METHOD PUBLIC Check_DT_TO_DINT_Max
VAR
	value : DT := DatatypeLimits.MAX_VALUE_OF_DT_WHICH_CAN_BE_HELD_IN_A_DINT;
	actual : DINT;
	converted : BOOL;
	equal : BOOL;
END_VAR
TEST('Check_DT_TO_DINT_Max');

// @TEST-RUN
converted := TryConvert_DT_TO_Destination(value, actual);
equal := actual = DT_TO_DINT(value);

// @TEST-ASSERT
AssertTrue(Condition := equal, Message := 'Did not convert DT to DINT correctly');
AssertTrue(Condition := converted, Message := 'Did not report DT to DINT conversion was successful');

TEST_FINISHED();
END_METHOD

METHOD PUBLIC Check_DT_TO_DINT_Min
VAR
	value : DT := DatatypeLimits.DT_MIN_VALUE;
	actual : DINT;
	converted : BOOL;
	equal : BOOL;
END_VAR
TEST('Check_DT_TO_DINT_Min');

// @TEST-RUN
converted := TryConvert_DT_TO_Destination(value, actual);
equal := actual = DT_TO_DINT(value);

// @TEST-ASSERT
AssertTrue(Condition := equal, Message := 'Did not convert DT to DINT correctly');
AssertTrue(Condition := converted, Message := 'Did not report DT to DINT conversion was successful');

TEST_FINISHED();
END_METHOD

METHOD PUBLIC Check_DT_TO_DINT_TooHigh
VAR
	value : DT := DatatypeLimits.DT_MAX_VALUE;
	actual : DINT;
	converted : BOOL;
END_VAR
TEST('Check_DT_TO_DINT_TooHigh');

// @TEST-RUN
converted := TryConvert_DT_TO_Destination(value, actual);

// @TEST-ASSERT
AssertFalse(Condition := converted, Message := 'Did not report DT to DINT conversion was prevented');

TEST_FINISHED();
END_METHOD

METHOD PUBLIC Check_DT_TO_DT_Max
VAR
	value : DT := DatatypeLimits.DT_MAX_VALUE;
	actual : DT;
	converted : BOOL;
	equal : BOOL;
END_VAR
TEST('Check_DT_TO_DT_Max');

// @TEST-RUN
converted := TryConvert_DT_TO_Destination(value, actual);
equal := actual = value;

// @TEST-ASSERT
AssertTrue(Condition := equal, Message := 'Did not convert DT to DT correctly');
AssertTrue(Condition := converted, Message := 'Did not report DT to DT conversion was successful');

TEST_FINISHED();
END_METHOD

METHOD PUBLIC Check_DT_TO_DT_Min
VAR
	value : DT := DatatypeLimits.DT_MIN_VALUE;
	actual : DT;
	converted : BOOL;
	equal : BOOL;
END_VAR
TEST('Check_DT_TO_DT_Min');

// @TEST-RUN
converted := TryConvert_DT_TO_Destination(value, actual);
equal := actual = value;

// @TEST-ASSERT
AssertTrue(Condition := equal, Message := 'Did not convert DT to DT correctly');
AssertTrue(Condition := converted, Message := 'Did not report DT to DT conversion was successful');

TEST_FINISHED();
END_METHOD

METHOD PUBLIC Check_DT_TO_DWORD_Max
VAR
	value : DT := DatatypeLimits.DT_MAX_VALUE;
	actual : DWORD;
	converted : BOOL;
	equal : BOOL;
END_VAR
TEST('Check_DT_TO_DWORD_Max');

// @TEST-RUN
converted := TryConvert_DT_TO_Destination(value, actual);
equal := actual = DT_TO_DWORD(value);

// @TEST-ASSERT
AssertTrue(Condition := equal, Message := 'Did not convert DT to DWORD correctly');
AssertTrue(Condition := converted, Message := 'Did not report DT to DWORD conversion was successful');

TEST_FINISHED();
END_METHOD

METHOD PUBLIC Check_DT_TO_DWORD_Min
VAR
	value : DT := DatatypeLimits.DT_MIN_VALUE;
	actual : DWORD;
	converted : BOOL;
	equal : BOOL;
END_VAR
TEST('Check_DT_TO_DWORD_Min');

// @TEST-RUN
converted := TryConvert_DT_TO_Destination(value, actual);
equal := actual = DT_TO_DWORD(value);

// @TEST-ASSERT
AssertTrue(Condition := equal, Message := 'Did not convert DT to DWORD correctly');
AssertTrue(Condition := converted, Message := 'Did not report DT to DWORD conversion was successful');

TEST_FINISHED();
END_METHOD

METHOD PUBLIC Check_DT_TO_INT_Max
VAR
	value : DT := DatatypeLimits.MAX_VALUE_OF_DT_WHICH_CAN_BE_HELD_IN_A_INT;
	actual : INT;
	converted : BOOL;
	equal : BOOL;
END_VAR
TEST('Check_DT_TO_INT_Max');

// @TEST-RUN
converted := TryConvert_DT_TO_Destination(value, actual);
equal := actual = DT_TO_INT(value);

// @TEST-ASSERT
AssertTrue(Condition := equal, Message := 'Did not convert DT to INT correctly');
AssertTrue(Condition := converted, Message := 'Did not report DT to INT conversion was successful');

TEST_FINISHED();
END_METHOD

METHOD PUBLIC Check_DT_TO_INT_Min
VAR
	value : DT := DatatypeLimits.DT_MIN_VALUE;
	actual : INT;
	converted : BOOL;
	equal : BOOL;
END_VAR
TEST('Check_DT_TO_INT_Min');

// @TEST-RUN
converted := TryConvert_DT_TO_Destination(value, actual);
equal := actual = DT_TO_INT(value);

// @TEST-ASSERT
AssertTrue(Condition := equal, Message := 'Did not convert DT to INT correctly');
AssertTrue(Condition := converted, Message := 'Did not report DT to INT conversion was successful');

TEST_FINISHED();
END_METHOD

METHOD PUBLIC Check_DT_TO_INT_TooHigh
VAR
	value : DT := DatatypeLimits.DT_MAX_VALUE;
	actual : INT;
	converted : BOOL;
END_VAR
TEST('Check_DT_TO_INT_TooHigh');

// @TEST-RUN
converted := TryConvert_DT_TO_Destination(value, actual);

// @TEST-ASSERT
AssertFalse(Condition := converted, Message := 'Did not report DT to INT conversion was prevented');

TEST_FINISHED();
END_METHOD

METHOD PUBLIC Check_DT_TO_LINT_Max
VAR
	value : DT := DatatypeLimits.DT_MAX_VALUE;
	actual : LINT;
	converted : BOOL;
	equal : BOOL;
END_VAR
TEST('Check_DT_TO_LINT_Max');

// @TEST-RUN
converted := TryConvert_DT_TO_Destination(value, actual);
equal := actual = DT_TO_LINT(value);

// @TEST-ASSERT
AssertTrue(Condition := equal, Message := 'Did not convert DT to LINT correctly');
AssertTrue(Condition := converted, Message := 'Did not report DT to LINT conversion was successful');

TEST_FINISHED();
END_METHOD

METHOD PUBLIC Check_DT_TO_LINT_Min
VAR
	value : DT := DatatypeLimits.DT_MIN_VALUE;
	actual : LINT;
	converted : BOOL;
	equal : BOOL;
END_VAR
TEST('Check_DT_TO_LINT_Min');

// @TEST-RUN
converted := TryConvert_DT_TO_Destination(value, actual);
equal := actual = DT_TO_LINT(value);

// @TEST-ASSERT
AssertTrue(Condition := equal, Message := 'Did not convert DT to LINT correctly');
AssertTrue(Condition := converted, Message := 'Did not report DT to LINT conversion was successful');

TEST_FINISHED();
END_METHOD

METHOD PUBLIC Check_DT_TO_LREAL_Max
VAR
	value : DT := DatatypeLimits.DT_MAX_VALUE;
	actual : LREAL;
	converted : BOOL;
	equal : BOOL;
END_VAR
TEST('Check_DT_TO_LREAL_Max');

// @TEST-RUN
converted := TryConvert_DT_TO_Destination(value, actual);
equal := actual = DT_TO_LREAL(value);

// @TEST-ASSERT
AssertTrue(Condition := equal, Message := 'Did not convert DT to LREAL correctly');
AssertTrue(Condition := converted, Message := 'Did not report DT to LREAL conversion was successful');

TEST_FINISHED();
END_METHOD

METHOD PUBLIC Check_DT_TO_LREAL_Min
VAR
	value : DT := DatatypeLimits.DT_MIN_VALUE;
	actual : LREAL;
	converted : BOOL;
	equal : BOOL;
END_VAR
TEST('Check_DT_TO_LREAL_Min');

// @TEST-RUN
converted := TryConvert_DT_TO_Destination(value, actual);
equal := actual = DT_TO_LREAL(value);

// @TEST-ASSERT
AssertTrue(Condition := equal, Message := 'Did not convert DT to LREAL correctly');
AssertTrue(Condition := converted, Message := 'Did not report DT to LREAL conversion was successful');

TEST_FINISHED();
END_METHOD

METHOD PUBLIC Check_DT_TO_LWORD_Max
VAR
	value : DT := DatatypeLimits.DT_MAX_VALUE;
	actual : LWORD;
	converted : BOOL;
	equal : BOOL;
END_VAR
TEST('Check_DT_TO_LWORD_Max');

// @TEST-RUN
converted := TryConvert_DT_TO_Destination(value, actual);
equal := actual = DT_TO_LWORD(value);

// @TEST-ASSERT
AssertTrue(Condition := equal, Message := 'Did not convert DT to LWORD correctly');
AssertTrue(Condition := converted, Message := 'Did not report DT to LWORD conversion was successful');

TEST_FINISHED();
END_METHOD

METHOD PUBLIC Check_DT_TO_LWORD_Min
VAR
	value : DT := DatatypeLimits.DT_MIN_VALUE;
	actual : LWORD;
	converted : BOOL;
	equal : BOOL;
END_VAR
TEST('Check_DT_TO_LWORD_Min');

// @TEST-RUN
converted := TryConvert_DT_TO_Destination(value, actual);
equal := actual = DT_TO_LWORD(value);

// @TEST-ASSERT
AssertTrue(Condition := equal, Message := 'Did not convert DT to LWORD correctly');
AssertTrue(Condition := converted, Message := 'Did not report DT to LWORD conversion was successful');

TEST_FINISHED();
END_METHOD

METHOD PUBLIC Check_DT_TO_REAL_Max
VAR
	value : DT := DatatypeLimits.DT_MAX_VALUE;
	actual : REAL;
	converted : BOOL;
	equal : BOOL;
END_VAR
TEST('Check_DT_TO_REAL_Max');

// @TEST-RUN
converted := TryConvert_DT_TO_Destination(value, actual);
equal := actual = DT_TO_REAL(value);

// @TEST-ASSERT
AssertTrue(Condition := equal, Message := 'Did not convert DT to REAL correctly');
AssertTrue(Condition := converted, Message := 'Did not report DT to REAL conversion was successful');

TEST_FINISHED();
END_METHOD

METHOD PUBLIC Check_DT_TO_REAL_Min
VAR
	value : DT := DatatypeLimits.DT_MIN_VALUE;
	actual : REAL;
	converted : BOOL;
	equal : BOOL;
END_VAR
TEST('Check_DT_TO_REAL_Min');

// @TEST-RUN
converted := TryConvert_DT_TO_Destination(value, actual);
equal := actual = DT_TO_REAL(value);

// @TEST-ASSERT
AssertTrue(Condition := equal, Message := 'Did not convert DT to REAL correctly');
AssertTrue(Condition := converted, Message := 'Did not report DT to REAL conversion was successful');

TEST_FINISHED();
END_METHOD

METHOD PUBLIC Check_DT_TO_SINT_Max
VAR
	value : DT := DatatypeLimits.MAX_VALUE_OF_DT_WHICH_CAN_BE_HELD_IN_A_SINT;
	actual : SINT;
	converted : BOOL;
	equal : BOOL;
END_VAR
TEST('Check_DT_TO_SINT_Max');

// @TEST-RUN
converted := TryConvert_DT_TO_Destination(value, actual);
equal := actual = DT_TO_SINT(value);

// @TEST-ASSERT
AssertTrue(Condition := equal, Message := 'Did not convert DT to SINT correctly');
AssertTrue(Condition := converted, Message := 'Did not report DT to SINT conversion was successful');

TEST_FINISHED();
END_METHOD

METHOD PUBLIC Check_DT_TO_SINT_Min
VAR
	value : DT := DatatypeLimits.DT_MIN_VALUE;
	actual : SINT;
	converted : BOOL;
	equal : BOOL;
END_VAR
TEST('Check_DT_TO_SINT_Min');

// @TEST-RUN
converted := TryConvert_DT_TO_Destination(value, actual);
equal := actual = DT_TO_SINT(value);

// @TEST-ASSERT
AssertTrue(Condition := equal, Message := 'Did not convert DT to SINT correctly');
AssertTrue(Condition := converted, Message := 'Did not report DT to SINT conversion was successful');

TEST_FINISHED();
END_METHOD

METHOD PUBLIC Check_DT_TO_SINT_TooHigh
VAR
	value : DT := DatatypeLimits.DT_MAX_VALUE;
	actual : SINT;
	converted : BOOL;
END_VAR
TEST('Check_DT_TO_SINT_TooHigh');

// @TEST-RUN
converted := TryConvert_DT_TO_Destination(value, actual);

// @TEST-ASSERT
AssertFalse(Condition := converted, Message := 'Did not report DT to SINT conversion was prevented');

TEST_FINISHED();
END_METHOD

METHOD PUBLIC Check_DT_TO_STRING_Max
VAR
	value : DT := DatatypeLimits.DT_MAX_VALUE;
	actual : STRING;
	converted : BOOL;
	equal : BOOL;
END_VAR
TEST('Check_DT_TO_STRING_Max');

// @TEST-RUN
converted := TryConvert_DT_TO_Destination(value, actual);
equal := actual = DT_TO_STRING(value);

// @TEST-ASSERT
AssertTrue(Condition := equal, Message := 'Did not convert DT to STRING correctly');
AssertTrue(Condition := converted, Message := 'Did not report DT to STRING conversion was successful');

TEST_FINISHED();
END_METHOD

METHOD PUBLIC Check_DT_TO_STRING_Min
VAR
	value : DT := DatatypeLimits.DT_MIN_VALUE;
	actual : STRING;
	converted : BOOL;
	equal : BOOL;
END_VAR
TEST('Check_DT_TO_STRING_Min');

// @TEST-RUN
converted := TryConvert_DT_TO_Destination(value, actual);
equal := actual = DT_TO_STRING(value);

// @TEST-ASSERT
AssertTrue(Condition := equal, Message := 'Did not convert DT to STRING correctly');
AssertTrue(Condition := converted, Message := 'Did not report DT to STRING conversion was successful');

TEST_FINISHED();
END_METHOD

METHOD PUBLIC Check_DT_TO_TIME_Max
VAR
	value : DT := DatatypeLimits.MAX_VALUE_OF_DT_WHICH_CAN_BE_HELD_IN_A_TIME;
	actual : TIME;
	converted : BOOL;
	equal : BOOL;
END_VAR
TEST('Check_DT_TO_TIME_Max');

// @TEST-RUN
converted := TryConvert_DT_TO_Destination(value, actual);
equal := actual = DT_TO_TIME(value);

// @TEST-ASSERT
AssertTrue(Condition := equal, Message := 'Did not convert DT to TIME correctly');
AssertTrue(Condition := converted, Message := 'Did not report DT to TIME conversion was successful');

TEST_FINISHED();
END_METHOD

METHOD PUBLIC Check_DT_TO_TIME_Min
VAR
	value : DT := DatatypeLimits.DT_MIN_VALUE;
	actual : TIME;
	converted : BOOL;
	equal : BOOL;
END_VAR
TEST('Check_DT_TO_TIME_Min');

// @TEST-RUN
converted := TryConvert_DT_TO_Destination(value, actual);
equal := actual = DT_TO_TIME(value);

// @TEST-ASSERT
AssertTrue(Condition := equal, Message := 'Did not convert DT to TIME correctly');
AssertTrue(Condition := converted, Message := 'Did not report DT to TIME conversion was successful');

TEST_FINISHED();
END_METHOD

METHOD PUBLIC Check_DT_TO_TIME_TooHigh
VAR
	value : DT := DatatypeLimits.DT_MAX_VALUE;
	actual : TIME;
	converted : BOOL;
END_VAR
TEST('Check_DT_TO_TIME_TooHigh');

// @TEST-RUN
converted := TryConvert_DT_TO_Destination(value, actual);

// @TEST-ASSERT
AssertFalse(Condition := converted, Message := 'Did not report DT to TIME conversion was prevented');

TEST_FINISHED();
END_METHOD

METHOD PUBLIC Check_DT_TO_TOD_Max
VAR
	value : DT := DatatypeLimits.MAX_VALUE_OF_DT_WHICH_CAN_BE_HELD_IN_A_TOD;
	actual : TOD;
	converted : BOOL;
	equal : BOOL;
END_VAR
TEST('Check_DT_TO_TOD_Max');

// @TEST-RUN
converted := TryConvert_DT_TO_Destination(value, actual);
equal := actual = DT_TO_TOD(value);

// @TEST-ASSERT
AssertTrue(Condition := equal, Message := 'Did not convert DT to TOD correctly');
AssertTrue(Condition := converted, Message := 'Did not report DT to TOD conversion was successful');

TEST_FINISHED();
END_METHOD

METHOD PUBLIC Check_DT_TO_TOD_Min
VAR
	value : DT := DatatypeLimits.DT_MIN_VALUE;
	actual : TOD;
	converted : BOOL;
	equal : BOOL;
END_VAR
TEST('Check_DT_TO_TOD_Min');

// @TEST-RUN
converted := TryConvert_DT_TO_Destination(value, actual);
equal := actual = DT_TO_TOD(value);

// @TEST-ASSERT
AssertTrue(Condition := equal, Message := 'Did not convert DT to TOD correctly');
AssertTrue(Condition := converted, Message := 'Did not report DT to TOD conversion was successful');

TEST_FINISHED();
END_METHOD

METHOD PUBLIC Check_DT_TO_TOD_TooHigh
VAR
	value : DT := DatatypeLimits.DT_MAX_VALUE;
	actual : TOD;
	converted : BOOL;
END_VAR
TEST('Check_DT_TO_TOD_TooHigh');

// @TEST-RUN
converted := TryConvert_DT_TO_Destination(value, actual);

// @TEST-ASSERT
AssertFalse(Condition := converted, Message := 'Did not report DT to TOD conversion was prevented');

TEST_FINISHED();
END_METHOD

METHOD PUBLIC Check_DT_TO_UDINT_Max
VAR
	value : DT := DatatypeLimits.DT_MAX_VALUE;
	actual : UDINT;
	converted : BOOL;
	equal : BOOL;
END_VAR
TEST('Check_DT_TO_UDINT_Max');

// @TEST-RUN
converted := TryConvert_DT_TO_Destination(value, actual);
equal := actual = DT_TO_UDINT(value);

// @TEST-ASSERT
AssertTrue(Condition := equal, Message := 'Did not convert DT to UDINT correctly');
AssertTrue(Condition := converted, Message := 'Did not report DT to UDINT conversion was successful');

TEST_FINISHED();
END_METHOD

METHOD PUBLIC Check_DT_TO_UDINT_Min
VAR
	value : DT := DatatypeLimits.DT_MIN_VALUE;
	actual : UDINT;
	converted : BOOL;
	equal : BOOL;
END_VAR
TEST('Check_DT_TO_UDINT_Min');

// @TEST-RUN
converted := TryConvert_DT_TO_Destination(value, actual);
equal := actual = DT_TO_UDINT(value);

// @TEST-ASSERT
AssertTrue(Condition := equal, Message := 'Did not convert DT to UDINT correctly');
AssertTrue(Condition := converted, Message := 'Did not report DT to UDINT conversion was successful');

TEST_FINISHED();
END_METHOD

METHOD PUBLIC Check_DT_TO_UINT_Max
VAR
	value : DT := DatatypeLimits.MAX_VALUE_OF_DT_WHICH_CAN_BE_HELD_IN_A_UINT;
	actual : UINT;
	converted : BOOL;
	equal : BOOL;
END_VAR
TEST('Check_DT_TO_UINT_Max');

// @TEST-RUN
converted := TryConvert_DT_TO_Destination(value, actual);
equal := actual = DT_TO_UINT(value);

// @TEST-ASSERT
AssertTrue(Condition := equal, Message := 'Did not convert DT to UINT correctly');
AssertTrue(Condition := converted, Message := 'Did not report DT to UINT conversion was successful');

TEST_FINISHED();
END_METHOD

METHOD PUBLIC Check_DT_TO_UINT_Min
VAR
	value : DT := DatatypeLimits.DT_MIN_VALUE;
	actual : UINT;
	converted : BOOL;
	equal : BOOL;
END_VAR
TEST('Check_DT_TO_UINT_Min');

// @TEST-RUN
converted := TryConvert_DT_TO_Destination(value, actual);
equal := actual = DT_TO_UINT(value);

// @TEST-ASSERT
AssertTrue(Condition := equal, Message := 'Did not convert DT to UINT correctly');
AssertTrue(Condition := converted, Message := 'Did not report DT to UINT conversion was successful');

TEST_FINISHED();
END_METHOD

METHOD PUBLIC Check_DT_TO_UINT_TooHigh
VAR
	value : DT := DatatypeLimits.DT_MAX_VALUE;
	actual : UINT;
	converted : BOOL;
END_VAR
TEST('Check_DT_TO_UINT_TooHigh');

// @TEST-RUN
converted := TryConvert_DT_TO_Destination(value, actual);

// @TEST-ASSERT
AssertFalse(Condition := converted, Message := 'Did not report DT to UINT conversion was prevented');

TEST_FINISHED();
END_METHOD

METHOD PUBLIC Check_DT_TO_ULINT_Max
VAR
	value : DT := DatatypeLimits.DT_MAX_VALUE;
	actual : ULINT;
	converted : BOOL;
	equal : BOOL;
END_VAR
TEST('Check_DT_TO_ULINT_Max');

// @TEST-RUN
converted := TryConvert_DT_TO_Destination(value, actual);
equal := actual = DT_TO_ULINT(value);

// @TEST-ASSERT
AssertTrue(Condition := equal, Message := 'Did not convert DT to ULINT correctly');
AssertTrue(Condition := converted, Message := 'Did not report DT to ULINT conversion was successful');

TEST_FINISHED();
END_METHOD

METHOD PUBLIC Check_DT_TO_ULINT_Min
VAR
	value : DT := DatatypeLimits.DT_MIN_VALUE;
	actual : ULINT;
	converted : BOOL;
	equal : BOOL;
END_VAR
TEST('Check_DT_TO_ULINT_Min');

// @TEST-RUN
converted := TryConvert_DT_TO_Destination(value, actual);
equal := actual = DT_TO_ULINT(value);

// @TEST-ASSERT
AssertTrue(Condition := equal, Message := 'Did not convert DT to ULINT correctly');
AssertTrue(Condition := converted, Message := 'Did not report DT to ULINT conversion was successful');

TEST_FINISHED();
END_METHOD

METHOD PUBLIC Check_DT_TO_USINT_Max
VAR
	value : DT := DatatypeLimits.MAX_VALUE_OF_DT_WHICH_CAN_BE_HELD_IN_A_USINT;
	actual : USINT;
	converted : BOOL;
	equal : BOOL;
END_VAR
TEST('Check_DT_TO_USINT_Max');

// @TEST-RUN
converted := TryConvert_DT_TO_Destination(value, actual);
equal := actual = DT_TO_USINT(value);

// @TEST-ASSERT
AssertTrue(Condition := equal, Message := 'Did not convert DT to USINT correctly');
AssertTrue(Condition := converted, Message := 'Did not report DT to USINT conversion was successful');

TEST_FINISHED();
END_METHOD

METHOD PUBLIC Check_DT_TO_USINT_Min
VAR
	value : DT := DatatypeLimits.DT_MIN_VALUE;
	actual : USINT;
	converted : BOOL;
	equal : BOOL;
END_VAR
TEST('Check_DT_TO_USINT_Min');

// @TEST-RUN
converted := TryConvert_DT_TO_Destination(value, actual);
equal := actual = DT_TO_USINT(value);

// @TEST-ASSERT
AssertTrue(Condition := equal, Message := 'Did not convert DT to USINT correctly');
AssertTrue(Condition := converted, Message := 'Did not report DT to USINT conversion was successful');

TEST_FINISHED();
END_METHOD

METHOD PUBLIC Check_DT_TO_USINT_TooHigh
VAR
	value : DT := DatatypeLimits.DT_MAX_VALUE;
	actual : USINT;
	converted : BOOL;
END_VAR
TEST('Check_DT_TO_USINT_TooHigh');

// @TEST-RUN
converted := TryConvert_DT_TO_Destination(value, actual);

// @TEST-ASSERT
AssertFalse(Condition := converted, Message := 'Did not report DT to USINT conversion was prevented');

TEST_FINISHED();
END_METHOD

METHOD PUBLIC Check_DT_TO_WORD_Max
VAR
	value : DT := DatatypeLimits.MAX_VALUE_OF_DT_WHICH_CAN_BE_HELD_IN_A_WORD;
	actual : WORD;
	converted : BOOL;
	equal : BOOL;
END_VAR
TEST('Check_DT_TO_WORD_Max');

// @TEST-RUN
converted := TryConvert_DT_TO_Destination(value, actual);
equal := actual = DT_TO_WORD(value);

// @TEST-ASSERT
AssertTrue(Condition := equal, Message := 'Did not convert DT to WORD correctly');
AssertTrue(Condition := converted, Message := 'Did not report DT to WORD conversion was successful');

TEST_FINISHED();
END_METHOD

METHOD PUBLIC Check_DT_TO_WORD_Min
VAR
	value : DT := DatatypeLimits.DT_MIN_VALUE;
	actual : WORD;
	converted : BOOL;
	equal : BOOL;
END_VAR
TEST('Check_DT_TO_WORD_Min');

// @TEST-RUN
converted := TryConvert_DT_TO_Destination(value, actual);
equal := actual = DT_TO_WORD(value);

// @TEST-ASSERT
AssertTrue(Condition := equal, Message := 'Did not convert DT to WORD correctly');
AssertTrue(Condition := converted, Message := 'Did not report DT to WORD conversion was successful');

TEST_FINISHED();
END_METHOD

METHOD PUBLIC Check_DT_TO_WORD_TooHigh
VAR
	value : DT := DatatypeLimits.DT_MAX_VALUE;
	actual : WORD;
	converted : BOOL;
END_VAR
TEST('Check_DT_TO_WORD_TooHigh');

// @TEST-RUN
converted := TryConvert_DT_TO_Destination(value, actual);

// @TEST-ASSERT
AssertFalse(Condition := converted, Message := 'Did not report DT to WORD conversion was prevented');

TEST_FINISHED();
END_METHOD

END_FUNCTION_BLOCK

// ---- mobject-converters/Tests/DWORD_TO_TestSuite.TcPOU
FUNCTION_BLOCK PUBLIC DWORD_TO_TestSuite EXTENDS TcUnit.FB_TestSuite
VAR
END_VAR

Check_DWORD_TO_BOOL_Max();
Check_DWORD_TO_BOOL_Min();
Check_DWORD_TO_BYTE_Max();
Check_DWORD_TO_BYTE_Min();
Check_DWORD_TO_BYTE_TooHigh();
Check_DWORD_TO_WORD_Max();
Check_DWORD_TO_WORD_Min();
Check_DWORD_TO_WORD_TooHigh();
Check_DWORD_TO_DWORD_Max();
Check_DWORD_TO_DWORD_Min();
Check_DWORD_TO_LWORD_Max();
Check_DWORD_TO_LWORD_Min();
Check_DWORD_TO_SINT_Max();
Check_DWORD_TO_SINT_Min();
Check_DWORD_TO_SINT_TooHigh();
Check_DWORD_TO_INT_Max();
Check_DWORD_TO_INT_Min();
Check_DWORD_TO_INT_TooHigh();
Check_DWORD_TO_DINT_Max();
Check_DWORD_TO_DINT_Min();
Check_DWORD_TO_DINT_TooHigh();
Check_DWORD_TO_LINT_Max();
Check_DWORD_TO_LINT_Min();
Check_DWORD_TO_USINT_Max();
Check_DWORD_TO_USINT_Min();
Check_DWORD_TO_USINT_TooHigh();
Check_DWORD_TO_UINT_Max();
Check_DWORD_TO_UINT_Min();
Check_DWORD_TO_UINT_TooHigh();
Check_DWORD_TO_UDINT_Max();
Check_DWORD_TO_UDINT_Min();
Check_DWORD_TO_ULINT_Max();
Check_DWORD_TO_ULINT_Min();
Check_DWORD_TO_REAL_Max();
Check_DWORD_TO_REAL_Min();
Check_DWORD_TO_LREAL_Max();
Check_DWORD_TO_LREAL_Min();
Check_DWORD_TO_TIME_Max();
Check_DWORD_TO_TIME_Min();
Check_DWORD_TO_TOD_Max();
Check_DWORD_TO_TOD_Min();
Check_DWORD_TO_TOD_TooHigh();
Check_DWORD_TO_DATE_Max();
Check_DWORD_TO_DATE_Min();
Check_DWORD_TO_DT_Max();
Check_DWORD_TO_DT_Min();
Check_DWORD_TO_STRING_Max();
Check_DWORD_TO_STRING_Min();

METHOD PUBLIC Check_DWORD_TO_BOOL_Max
VAR
	value : DWORD := DatatypeLimits.DWORD_MAX_VALUE;
	actual : BOOL;
	converted : BOOL;
	equal : BOOL;
END_VAR
TEST('Check_DWORD_TO_BOOL_Max');

// @TEST-RUN
converted := TryConvert_DWORD_TO_Destination(value, actual);
equal := actual = DWORD_TO_BOOL(value);

// @TEST-ASSERT
AssertTrue(Condition := equal, Message := 'Did not convert DWORD to BOOL correctly');
AssertTrue(Condition := converted, Message := 'Did not report DWORD to BOOL conversion was successful');

TEST_FINISHED();
END_METHOD

METHOD PUBLIC Check_DWORD_TO_BOOL_Min
VAR
	value : DWORD := DatatypeLimits.DWORD_MIN_VALUE;
	actual : BOOL;
	converted : BOOL;
	equal : BOOL;
END_VAR
TEST('Check_DWORD_TO_BOOL_Min');

// @TEST-RUN
converted := TryConvert_DWORD_TO_Destination(value, actual);
equal := actual = DWORD_TO_BOOL(value);

// @TEST-ASSERT
AssertTrue(Condition := equal, Message := 'Did not convert DWORD to BOOL correctly');
AssertTrue(Condition := converted, Message := 'Did not report DWORD to BOOL conversion was successful');

TEST_FINISHED();
END_METHOD

METHOD PUBLIC Check_DWORD_TO_BYTE_Max
VAR
	value : DWORD := DatatypeLimits.MAX_VALUE_OF_DWORD_WHICH_CAN_BE_HELD_IN_A_BYTE;
	actual : BYTE;
	converted : BOOL;
	equal : BOOL;
END_VAR
TEST('Check_DWORD_TO_BYTE_Max');

// @TEST-RUN
converted := TryConvert_DWORD_TO_Destination(value, actual);
equal := actual = DWORD_TO_BYTE(value);

// @TEST-ASSERT
AssertTrue(Condition := equal, Message := 'Did not convert DWORD to BYTE correctly');
AssertTrue(Condition := converted, Message := 'Did not report DWORD to BYTE conversion was successful');

TEST_FINISHED();
END_METHOD

METHOD PUBLIC Check_DWORD_TO_BYTE_Min
VAR
	value : DWORD := DatatypeLimits.DWORD_MIN_VALUE;
	actual : BYTE;
	converted : BOOL;
	equal : BOOL;
END_VAR
TEST('Check_DWORD_TO_BYTE_Min');

// @TEST-RUN
converted := TryConvert_DWORD_TO_Destination(value, actual);
equal := actual = DWORD_TO_BYTE(value);

// @TEST-ASSERT
AssertTrue(Condition := equal, Message := 'Did not convert DWORD to BYTE correctly');
AssertTrue(Condition := converted, Message := 'Did not report DWORD to BYTE conversion was successful');

TEST_FINISHED();
END_METHOD

METHOD PUBLIC Check_DWORD_TO_BYTE_TooHigh
VAR
	value : DWORD := DatatypeLimits.DWORD_MAX_VALUE;
	actual : BYTE;
	converted : BOOL;
END_VAR
TEST('Check_DWORD_TO_BYTE_TooHigh');

// @TEST-RUN
converted := TryConvert_DWORD_TO_Destination(value, actual);

// @TEST-ASSERT
AssertFalse(Condition := converted, Message := 'Did not report DWORD to BYTE conversion was prevented');

TEST_FINISHED();
END_METHOD

METHOD PUBLIC Check_DWORD_TO_DATE_Max
VAR
	value : DWORD := DatatypeLimits.DWORD_MAX_VALUE;
	actual : DATE;
	converted : BOOL;
	equal : BOOL;
END_VAR
TEST('Check_DWORD_TO_DATE_Max');

// @TEST-RUN
converted := TryConvert_DWORD_TO_Destination(value, actual);
equal := actual = DWORD_TO_DATE(value);

// @TEST-ASSERT
AssertTrue(Condition := equal, Message := 'Did not convert DWORD to DATE correctly');
AssertTrue(Condition := converted, Message := 'Did not report DWORD to DATE conversion was successful');

TEST_FINISHED();
END_METHOD

METHOD PUBLIC Check_DWORD_TO_DATE_Min
VAR
	value : DWORD := DatatypeLimits.DWORD_MIN_VALUE;
	actual : DATE;
	converted : BOOL;
	equal : BOOL;
END_VAR
TEST('Check_DWORD_TO_DATE_Min');

// @TEST-RUN
converted := TryConvert_DWORD_TO_Destination(value, actual);
equal := actual = DWORD_TO_DATE(value);

// @TEST-ASSERT
AssertTrue(Condition := equal, Message := 'Did not convert DWORD to DATE correctly');
AssertTrue(Condition := converted, Message := 'Did not report DWORD to DATE conversion was successful');

TEST_FINISHED();
END_METHOD

METHOD PUBLIC Check_DWORD_TO_DINT_Max
VAR
	value : DWORD := DatatypeLimits.MAX_VALUE_OF_DWORD_WHICH_CAN_BE_HELD_IN_A_DINT;
	actual : DINT;
	converted : BOOL;
	equal : BOOL;
END_VAR
TEST('Check_DWORD_TO_DINT_Max');

// @TEST-RUN
converted := TryConvert_DWORD_TO_Destination(value, actual);
equal := actual = DWORD_TO_DINT(value);

// @TEST-ASSERT
AssertTrue(Condition := equal, Message := 'Did not convert DWORD to DINT correctly');
AssertTrue(Condition := converted, Message := 'Did not report DWORD to DINT conversion was successful');

TEST_FINISHED();
END_METHOD

METHOD PUBLIC Check_DWORD_TO_DINT_Min
VAR
	value : DWORD := DatatypeLimits.DWORD_MIN_VALUE;
	actual : DINT;
	converted : BOOL;
	equal : BOOL;
END_VAR
TEST('Check_DWORD_TO_DINT_Min');

// @TEST-RUN
converted := TryConvert_DWORD_TO_Destination(value, actual);
equal := actual = DWORD_TO_DINT(value);

// @TEST-ASSERT
AssertTrue(Condition := equal, Message := 'Did not convert DWORD to DINT correctly');
AssertTrue(Condition := converted, Message := 'Did not report DWORD to DINT conversion was successful');

TEST_FINISHED();
END_METHOD

METHOD PUBLIC Check_DWORD_TO_DINT_TooHigh
VAR
	value : DWORD := DatatypeLimits.DWORD_MAX_VALUE;
	actual : DINT;
	converted : BOOL;
END_VAR
TEST('Check_DWORD_TO_DINT_TooHigh');

// @TEST-RUN
converted := TryConvert_DWORD_TO_Destination(value, actual);

// @TEST-ASSERT
AssertFalse(Condition := converted, Message := 'Did not report DWORD to DINT conversion was prevented');

TEST_FINISHED();
END_METHOD

METHOD PUBLIC Check_DWORD_TO_DT_Max
VAR
	value : DWORD := DatatypeLimits.DWORD_MAX_VALUE;
	actual : DT;
	converted : BOOL;
	equal : BOOL;
END_VAR
TEST('Check_DWORD_TO_DT_Max');

// @TEST-RUN
converted := TryConvert_DWORD_TO_Destination(value, actual);
equal := actual = DWORD_TO_DT(value);

// @TEST-ASSERT
AssertTrue(Condition := equal, Message := 'Did not convert DWORD to DT correctly');
AssertTrue(Condition := converted, Message := 'Did not report DWORD to DT conversion was successful');

TEST_FINISHED();
END_METHOD

METHOD PUBLIC Check_DWORD_TO_DT_Min
VAR
	value : DWORD := DatatypeLimits.DWORD_MIN_VALUE;
	actual : DT;
	converted : BOOL;
	equal : BOOL;
END_VAR
TEST('Check_DWORD_TO_DT_Min');

// @TEST-RUN
converted := TryConvert_DWORD_TO_Destination(value, actual);
equal := actual = DWORD_TO_DT(value);

// @TEST-ASSERT
AssertTrue(Condition := equal, Message := 'Did not convert DWORD to DT correctly');
AssertTrue(Condition := converted, Message := 'Did not report DWORD to DT conversion was successful');

TEST_FINISHED();
END_METHOD

METHOD PUBLIC Check_DWORD_TO_DWORD_Max
VAR
	value : DWORD := DatatypeLimits.DWORD_MAX_VALUE;
	actual : DWORD;
	converted : BOOL;
	equal : BOOL;
END_VAR
TEST('Check_DWORD_TO_DWORD_Max');

// @TEST-RUN
converted := TryConvert_DWORD_TO_Destination(value, actual);
equal := actual = value;

// @TEST-ASSERT
AssertTrue(Condition := equal, Message := 'Did not convert DWORD to DWORD correctly');
AssertTrue(Condition := converted, Message := 'Did not report DWORD to DWORD conversion was successful');

TEST_FINISHED();
END_METHOD

METHOD PUBLIC Check_DWORD_TO_DWORD_Min
VAR
	value : DWORD := DatatypeLimits.DWORD_MIN_VALUE;
	actual : DWORD;
	converted : BOOL;
	equal : BOOL;
END_VAR
TEST('Check_DWORD_TO_DWORD_Min');

// @TEST-RUN
converted := TryConvert_DWORD_TO_Destination(value, actual);
equal := actual = value;

// @TEST-ASSERT
AssertTrue(Condition := equal, Message := 'Did not convert DWORD to DWORD correctly');
AssertTrue(Condition := converted, Message := 'Did not report DWORD to DWORD conversion was successful');

TEST_FINISHED();
END_METHOD

METHOD PUBLIC Check_DWORD_TO_INT_Max
VAR
	value : DWORD := DatatypeLimits.MAX_VALUE_OF_DWORD_WHICH_CAN_BE_HELD_IN_A_INT;
	actual : INT;
	converted : BOOL;
	equal : BOOL;
END_VAR
TEST('Check_DWORD_TO_INT_Max');

// @TEST-RUN
converted := TryConvert_DWORD_TO_Destination(value, actual);
equal := actual = DWORD_TO_INT(value);

// @TEST-ASSERT
AssertTrue(Condition := equal, Message := 'Did not convert DWORD to INT correctly');
AssertTrue(Condition := converted, Message := 'Did not report DWORD to INT conversion was successful');

TEST_FINISHED();
END_METHOD

METHOD PUBLIC Check_DWORD_TO_INT_Min
VAR
	value : DWORD := DatatypeLimits.DWORD_MIN_VALUE;
	actual : INT;
	converted : BOOL;
	equal : BOOL;
END_VAR
TEST('Check_DWORD_TO_INT_Min');

// @TEST-RUN
converted := TryConvert_DWORD_TO_Destination(value, actual);
equal := actual = DWORD_TO_INT(value);

// @TEST-ASSERT
AssertTrue(Condition := equal, Message := 'Did not convert DWORD to INT correctly');
AssertTrue(Condition := converted, Message := 'Did not report DWORD to INT conversion was successful');

TEST_FINISHED();
END_METHOD

METHOD PUBLIC Check_DWORD_TO_INT_TooHigh
VAR
	value : DWORD := DatatypeLimits.DWORD_MAX_VALUE;
	actual : INT;
	converted : BOOL;
END_VAR
TEST('Check_DWORD_TO_INT_TooHigh');

// @TEST-RUN
converted := TryConvert_DWORD_TO_Destination(value, actual);

// @TEST-ASSERT
AssertFalse(Condition := converted, Message := 'Did not report DWORD to INT conversion was prevented');

TEST_FINISHED();
END_METHOD

METHOD PUBLIC Check_DWORD_TO_LINT_Max
VAR
	value : DWORD := DatatypeLimits.DWORD_MAX_VALUE;
	actual : LINT;
	converted : BOOL;
	equal : BOOL;
END_VAR
TEST('Check_DWORD_TO_LINT_Max');

// @TEST-RUN
converted := TryConvert_DWORD_TO_Destination(value, actual);
equal := actual = DWORD_TO_LINT(value);

// @TEST-ASSERT
AssertTrue(Condition := equal, Message := 'Did not convert DWORD to LINT correctly');
AssertTrue(Condition := converted, Message := 'Did not report DWORD to LINT conversion was successful');

TEST_FINISHED();
END_METHOD

METHOD PUBLIC Check_DWORD_TO_LINT_Min
VAR
	value : DWORD := DatatypeLimits.DWORD_MIN_VALUE;
	actual : LINT;
	converted : BOOL;
	equal : BOOL;
END_VAR
TEST('Check_DWORD_TO_LINT_Min');

// @TEST-RUN
converted := TryConvert_DWORD_TO_Destination(value, actual);
equal := actual = DWORD_TO_LINT(value);

// @TEST-ASSERT
AssertTrue(Condition := equal, Message := 'Did not convert DWORD to LINT correctly');
AssertTrue(Condition := converted, Message := 'Did not report DWORD to LINT conversion was successful');

TEST_FINISHED();
END_METHOD

METHOD PUBLIC Check_DWORD_TO_LREAL_Max
VAR
	value : DWORD := DatatypeLimits.DWORD_MAX_VALUE;
	actual : LREAL;
	converted : BOOL;
	equal : BOOL;
END_VAR
TEST('Check_DWORD_TO_LREAL_Max');

// @TEST-RUN
converted := TryConvert_DWORD_TO_Destination(value, actual);
equal := actual = DWORD_TO_LREAL(value);

// @TEST-ASSERT
AssertTrue(Condition := equal, Message := 'Did not convert DWORD to LREAL correctly');
AssertTrue(Condition := converted, Message := 'Did not report DWORD to LREAL conversion was successful');

TEST_FINISHED();
END_METHOD

METHOD PUBLIC Check_DWORD_TO_LREAL_Min
VAR
	value : DWORD := DatatypeLimits.DWORD_MIN_VALUE;
	actual : LREAL;
	converted : BOOL;
	equal : BOOL;
END_VAR
TEST('Check_DWORD_TO_LREAL_Min');

// @TEST-RUN
converted := TryConvert_DWORD_TO_Destination(value, actual);
equal := actual = DWORD_TO_LREAL(value);

// @TEST-ASSERT
AssertTrue(Condition := equal, Message := 'Did not convert DWORD to LREAL correctly');
AssertTrue(Condition := converted, Message := 'Did not report DWORD to LREAL conversion was successful');

TEST_FINISHED();
END_METHOD

METHOD PUBLIC Check_DWORD_TO_LWORD_Max
VAR
	value : DWORD := DatatypeLimits.DWORD_MAX_VALUE;
	actual : LWORD;
	converted : BOOL;
	equal : BOOL;
END_VAR
TEST('Check_DWORD_TO_LWORD_Max');

// @TEST-RUN
converted := TryConvert_DWORD_TO_Destination(value, actual);
equal := actual = DWORD_TO_LWORD(value);

// @TEST-ASSERT
AssertTrue(Condition := equal, Message := 'Did not convert DWORD to LWORD correctly');
AssertTrue(Condition := converted, Message := 'Did not report DWORD to LWORD conversion was successful');

TEST_FINISHED();
END_METHOD

METHOD PUBLIC Check_DWORD_TO_LWORD_Min
VAR
	value : DWORD := DatatypeLimits.DWORD_MIN_VALUE;
	actual : LWORD;
	converted : BOOL;
	equal : BOOL;
END_VAR
TEST('Check_DWORD_TO_LWORD_Min');

// @TEST-RUN
converted := TryConvert_DWORD_TO_Destination(value, actual);
equal := actual = DWORD_TO_LWORD(value);

// @TEST-ASSERT
AssertTrue(Condition := equal, Message := 'Did not convert DWORD to LWORD correctly');
AssertTrue(Condition := converted, Message := 'Did not report DWORD to LWORD conversion was successful');

TEST_FINISHED();
END_METHOD

METHOD PUBLIC Check_DWORD_TO_REAL_Max
VAR
	value : DWORD := DatatypeLimits.DWORD_MAX_VALUE;
	actual : REAL;
	converted : BOOL;
	equal : BOOL;
END_VAR
TEST('Check_DWORD_TO_REAL_Max');

// @TEST-RUN
converted := TryConvert_DWORD_TO_Destination(value, actual);
equal := actual = DWORD_TO_REAL(value);

// @TEST-ASSERT
AssertTrue(Condition := equal, Message := 'Did not convert DWORD to REAL correctly');
AssertTrue(Condition := converted, Message := 'Did not report DWORD to REAL conversion was successful');

TEST_FINISHED();
END_METHOD

METHOD PUBLIC Check_DWORD_TO_REAL_Min
VAR
	value : DWORD := DatatypeLimits.DWORD_MIN_VALUE;
	actual : REAL;
	converted : BOOL;
	equal : BOOL;
END_VAR
TEST('Check_DWORD_TO_REAL_Min');

// @TEST-RUN
converted := TryConvert_DWORD_TO_Destination(value, actual);
equal := actual = DWORD_TO_REAL(value);

// @TEST-ASSERT
AssertTrue(Condition := equal, Message := 'Did not convert DWORD to REAL correctly');
AssertTrue(Condition := converted, Message := 'Did not report DWORD to REAL conversion was successful');

TEST_FINISHED();
END_METHOD

METHOD PUBLIC Check_DWORD_TO_SINT_Max
VAR
	value : DWORD := DatatypeLimits.MAX_VALUE_OF_DWORD_WHICH_CAN_BE_HELD_IN_A_SINT;
	actual : SINT;
	converted : BOOL;
	equal : BOOL;
END_VAR
TEST('Check_DWORD_TO_SINT_Max');

// @TEST-RUN
converted := TryConvert_DWORD_TO_Destination(value, actual);
equal := actual = DWORD_TO_SINT(value);

// @TEST-ASSERT
AssertTrue(Condition := equal, Message := 'Did not convert DWORD to SINT correctly');
AssertTrue(Condition := converted, Message := 'Did not report DWORD to SINT conversion was successful');

TEST_FINISHED();
END_METHOD

METHOD PUBLIC Check_DWORD_TO_SINT_Min
VAR
	value : DWORD := DatatypeLimits.DWORD_MIN_VALUE;
	actual : SINT;
	converted : BOOL;
	equal : BOOL;
END_VAR
TEST('Check_DWORD_TO_SINT_Min');

// @TEST-RUN
converted := TryConvert_DWORD_TO_Destination(value, actual);
equal := actual = DWORD_TO_SINT(value);

// @TEST-ASSERT
AssertTrue(Condition := equal, Message := 'Did not convert DWORD to SINT correctly');
AssertTrue(Condition := converted, Message := 'Did not report DWORD to SINT conversion was successful');

TEST_FINISHED();
END_METHOD

METHOD PUBLIC Check_DWORD_TO_SINT_TooHigh
VAR
	value : DWORD := DatatypeLimits.DWORD_MAX_VALUE;
	actual : SINT;
	converted : BOOL;
END_VAR
TEST('Check_DWORD_TO_SINT_TooHigh');

// @TEST-RUN
converted := TryConvert_DWORD_TO_Destination(value, actual);

// @TEST-ASSERT
AssertFalse(Condition := converted, Message := 'Did not report DWORD to SINT conversion was prevented');

TEST_FINISHED();
END_METHOD

METHOD PUBLIC Check_DWORD_TO_STRING_Max
VAR
	value : DWORD := DatatypeLimits.DWORD_MAX_VALUE;
	actual : STRING;
	converted : BOOL;
	equal : BOOL;
END_VAR
TEST('Check_DWORD_TO_STRING_Max');

// @TEST-RUN
converted := TryConvert_DWORD_TO_Destination(value, actual);
equal := actual = DWORD_TO_STRING(value);

// @TEST-ASSERT
AssertTrue(Condition := equal, Message := 'Did not convert DWORD to STRING correctly');
AssertTrue(Condition := converted, Message := 'Did not report DWORD to STRING conversion was successful');

TEST_FINISHED();
END_METHOD

METHOD PUBLIC Check_DWORD_TO_STRING_Min
VAR
	value : DWORD := DatatypeLimits.DWORD_MIN_VALUE;
	actual : STRING;
	converted : BOOL;
	equal : BOOL;
END_VAR
TEST('Check_DWORD_TO_STRING_Min');

// @TEST-RUN
converted := TryConvert_DWORD_TO_Destination(value, actual);
equal := actual = DWORD_TO_STRING(value);

// @TEST-ASSERT
AssertTrue(Condition := equal, Message := 'Did not convert DWORD to STRING correctly');
AssertTrue(Condition := converted, Message := 'Did not report DWORD to STRING conversion was successful');

TEST_FINISHED();
END_METHOD

METHOD PUBLIC Check_DWORD_TO_TIME_Max
VAR
	value : DWORD := DatatypeLimits.DWORD_MAX_VALUE;
	actual : TIME;
	converted : BOOL;
	equal : BOOL;
END_VAR
TEST('Check_DWORD_TO_TIME_Max');

// @TEST-RUN
converted := TryConvert_DWORD_TO_Destination(value, actual);
equal := actual = DWORD_TO_TIME(value);

// @TEST-ASSERT
AssertTrue(Condition := equal, Message := 'Did not convert DWORD to TIME correctly');
AssertTrue(Condition := converted, Message := 'Did not report DWORD to TIME conversion was successful');

TEST_FINISHED();
END_METHOD

METHOD PUBLIC Check_DWORD_TO_TIME_Min
VAR
	value : DWORD := DatatypeLimits.DWORD_MIN_VALUE;
	actual : TIME;
	converted : BOOL;
	equal : BOOL;
END_VAR
TEST('Check_DWORD_TO_TIME_Min');

// @TEST-RUN
converted := TryConvert_DWORD_TO_Destination(value, actual);
equal := actual = DWORD_TO_TIME(value);

// @TEST-ASSERT
AssertTrue(Condition := equal, Message := 'Did not convert DWORD to TIME correctly');
AssertTrue(Condition := converted, Message := 'Did not report DWORD to TIME conversion was successful');

TEST_FINISHED();
END_METHOD

METHOD PUBLIC Check_DWORD_TO_TOD_Max
VAR
	value : DWORD := DatatypeLimits.MAX_VALUE_OF_DWORD_WHICH_CAN_BE_HELD_IN_A_TOD;
	actual : TOD;
	converted : BOOL;
	equal : BOOL;
END_VAR
TEST('Check_DWORD_TO_TOD_Max');

// @TEST-RUN
converted := TryConvert_DWORD_TO_Destination(value, actual);
equal := actual = DWORD_TO_TOD(value);

// @TEST-ASSERT
AssertTrue(Condition := equal, Message := 'Did not convert DWORD to TOD correctly');
AssertTrue(Condition := converted, Message := 'Did not report DWORD to TOD conversion was successful');

TEST_FINISHED();
END_METHOD

METHOD PUBLIC Check_DWORD_TO_TOD_Min
VAR
	value : DWORD := DatatypeLimits.DWORD_MIN_VALUE;
	actual : TOD;
	converted : BOOL;
	equal : BOOL;
END_VAR
TEST('Check_DWORD_TO_TOD_Min');

// @TEST-RUN
converted := TryConvert_DWORD_TO_Destination(value, actual);
equal := actual = DWORD_TO_TOD(value);

// @TEST-ASSERT
AssertTrue(Condition := equal, Message := 'Did not convert DWORD to TOD correctly');
AssertTrue(Condition := converted, Message := 'Did not report DWORD to TOD conversion was successful');

TEST_FINISHED();
END_METHOD

METHOD PUBLIC Check_DWORD_TO_TOD_TooHigh
VAR
	value : DWORD := DatatypeLimits.DWORD_MAX_VALUE;
	actual : TOD;
	converted : BOOL;
END_VAR
TEST('Check_DWORD_TO_TOD_TooHigh');

// @TEST-RUN
converted := TryConvert_DWORD_TO_Destination(value, actual);

// @TEST-ASSERT
AssertFalse(Condition := converted, Message := 'Did not report DWORD to TOD conversion was prevented');

TEST_FINISHED();
END_METHOD

METHOD PUBLIC Check_DWORD_TO_UDINT_Max
VAR
	value : DWORD := DatatypeLimits.DWORD_MAX_VALUE;
	actual : UDINT;
	converted : BOOL;
	equal : BOOL;
END_VAR
TEST('Check_DWORD_TO_UDINT_Max');

// @TEST-RUN
converted := TryConvert_DWORD_TO_Destination(value, actual);
equal := actual = DWORD_TO_UDINT(value);

// @TEST-ASSERT
AssertTrue(Condition := equal, Message := 'Did not convert DWORD to UDINT correctly');
AssertTrue(Condition := converted, Message := 'Did not report DWORD to UDINT conversion was successful');

TEST_FINISHED();
END_METHOD

METHOD PUBLIC Check_DWORD_TO_UDINT_Min
VAR
	value : DWORD := DatatypeLimits.DWORD_MIN_VALUE;
	actual : UDINT;
	converted : BOOL;
	equal : BOOL;
END_VAR
TEST('Check_DWORD_TO_UDINT_Min');

// @TEST-RUN
converted := TryConvert_DWORD_TO_Destination(value, actual);
equal := actual = DWORD_TO_UDINT(value);

// @TEST-ASSERT
AssertTrue(Condition := equal, Message := 'Did not convert DWORD to UDINT correctly');
AssertTrue(Condition := converted, Message := 'Did not report DWORD to UDINT conversion was successful');

TEST_FINISHED();
END_METHOD

METHOD PUBLIC Check_DWORD_TO_UINT_Max
VAR
	value : DWORD := DatatypeLimits.MAX_VALUE_OF_DWORD_WHICH_CAN_BE_HELD_IN_A_UINT;
	actual : UINT;
	converted : BOOL;
	equal : BOOL;
END_VAR
TEST('Check_DWORD_TO_UINT_Max');

// @TEST-RUN
converted := TryConvert_DWORD_TO_Destination(value, actual);
equal := actual = DWORD_TO_UINT(value);

// @TEST-ASSERT
AssertTrue(Condition := equal, Message := 'Did not convert DWORD to UINT correctly');
AssertTrue(Condition := converted, Message := 'Did not report DWORD to UINT conversion was successful');

TEST_FINISHED();
END_METHOD

METHOD PUBLIC Check_DWORD_TO_UINT_Min
VAR
	value : DWORD := DatatypeLimits.DWORD_MIN_VALUE;
	actual : UINT;
	converted : BOOL;
	equal : BOOL;
END_VAR
TEST('Check_DWORD_TO_UINT_Min');

// @TEST-RUN
converted := TryConvert_DWORD_TO_Destination(value, actual);
equal := actual = DWORD_TO_UINT(value);

// @TEST-ASSERT
AssertTrue(Condition := equal, Message := 'Did not convert DWORD to UINT correctly');
AssertTrue(Condition := converted, Message := 'Did not report DWORD to UINT conversion was successful');

TEST_FINISHED();
END_METHOD

METHOD PUBLIC Check_DWORD_TO_UINT_TooHigh
VAR
	value : DWORD := DatatypeLimits.DWORD_MAX_VALUE;
	actual : UINT;
	converted : BOOL;
END_VAR
TEST('Check_DWORD_TO_UINT_TooHigh');

// @TEST-RUN
converted := TryConvert_DWORD_TO_Destination(value, actual);

// @TEST-ASSERT
AssertFalse(Condition := converted, Message := 'Did not report DWORD to UINT conversion was prevented');

TEST_FINISHED();
END_METHOD

METHOD PUBLIC Check_DWORD_TO_ULINT_Max
VAR
	value : DWORD := DatatypeLimits.DWORD_MAX_VALUE;
	actual : ULINT;
	converted : BOOL;
	equal : BOOL;
END_VAR
TEST('Check_DWORD_TO_ULINT_Max');

// @TEST-RUN
converted := TryConvert_DWORD_TO_Destination(value, actual);
equal := actual = DWORD_TO_ULINT(value);

// @TEST-ASSERT
AssertTrue(Condition := equal, Message := 'Did not convert DWORD to ULINT correctly');
AssertTrue(Condition := converted, Message := 'Did not report DWORD to ULINT conversion was successful');

TEST_FINISHED();
END_METHOD

METHOD PUBLIC Check_DWORD_TO_ULINT_Min
VAR
	value : DWORD := DatatypeLimits.DWORD_MIN_VALUE;
	actual : ULINT;
	converted : BOOL;
	equal : BOOL;
END_VAR
TEST('Check_DWORD_TO_ULINT_Min');

// @TEST-RUN
converted := TryConvert_DWORD_TO_Destination(value, actual);
equal := actual = DWORD_TO_ULINT(value);

// @TEST-ASSERT
AssertTrue(Condition := equal, Message := 'Did not convert DWORD to ULINT correctly');
AssertTrue(Condition := converted, Message := 'Did not report DWORD to ULINT conversion was successful');

TEST_FINISHED();
END_METHOD

METHOD PUBLIC Check_DWORD_TO_USINT_Max
VAR
	value : DWORD := DatatypeLimits.MAX_VALUE_OF_DWORD_WHICH_CAN_BE_HELD_IN_A_USINT;
	actual : USINT;
	converted : BOOL;
	equal : BOOL;
END_VAR
TEST('Check_DWORD_TO_USINT_Max');

// @TEST-RUN
converted := TryConvert_DWORD_TO_Destination(value, actual);
equal := actual = DWORD_TO_USINT(value);

// @TEST-ASSERT
AssertTrue(Condition := equal, Message := 'Did not convert DWORD to USINT correctly');
AssertTrue(Condition := converted, Message := 'Did not report DWORD to USINT conversion was successful');

TEST_FINISHED();
END_METHOD

METHOD PUBLIC Check_DWORD_TO_USINT_Min
VAR
	value : DWORD := DatatypeLimits.DWORD_MIN_VALUE;
	actual : USINT;
	converted : BOOL;
	equal : BOOL;
END_VAR
TEST('Check_DWORD_TO_USINT_Min');

// @TEST-RUN
converted := TryConvert_DWORD_TO_Destination(value, actual);
equal := actual = DWORD_TO_USINT(value);

// @TEST-ASSERT
AssertTrue(Condition := equal, Message := 'Did not convert DWORD to USINT correctly');
AssertTrue(Condition := converted, Message := 'Did not report DWORD to USINT conversion was successful');

TEST_FINISHED();
END_METHOD

METHOD PUBLIC Check_DWORD_TO_USINT_TooHigh
VAR
	value : DWORD := DatatypeLimits.DWORD_MAX_VALUE;
	actual : USINT;
	converted : BOOL;
END_VAR
TEST('Check_DWORD_TO_USINT_TooHigh');

// @TEST-RUN
converted := TryConvert_DWORD_TO_Destination(value, actual);

// @TEST-ASSERT
AssertFalse(Condition := converted, Message := 'Did not report DWORD to USINT conversion was prevented');

TEST_FINISHED();
END_METHOD

METHOD PUBLIC Check_DWORD_TO_WORD_Max
VAR
	value : DWORD := DatatypeLimits.MAX_VALUE_OF_DWORD_WHICH_CAN_BE_HELD_IN_A_WORD;
	actual : WORD;
	converted : BOOL;
	equal : BOOL;
END_VAR
TEST('Check_DWORD_TO_WORD_Max');

// @TEST-RUN
converted := TryConvert_DWORD_TO_Destination(value, actual);
equal := actual = DWORD_TO_WORD(value);

// @TEST-ASSERT
AssertTrue(Condition := equal, Message := 'Did not convert DWORD to WORD correctly');
AssertTrue(Condition := converted, Message := 'Did not report DWORD to WORD conversion was successful');

TEST_FINISHED();
END_METHOD

METHOD PUBLIC Check_DWORD_TO_WORD_Min
VAR
	value : DWORD := DatatypeLimits.DWORD_MIN_VALUE;
	actual : WORD;
	converted : BOOL;
	equal : BOOL;
END_VAR
TEST('Check_DWORD_TO_WORD_Min');

// @TEST-RUN
converted := TryConvert_DWORD_TO_Destination(value, actual);
equal := actual = DWORD_TO_WORD(value);

// @TEST-ASSERT
AssertTrue(Condition := equal, Message := 'Did not convert DWORD to WORD correctly');
AssertTrue(Condition := converted, Message := 'Did not report DWORD to WORD conversion was successful');

TEST_FINISHED();
END_METHOD

METHOD PUBLIC Check_DWORD_TO_WORD_TooHigh
VAR
	value : DWORD := DatatypeLimits.DWORD_MAX_VALUE;
	actual : WORD;
	converted : BOOL;
END_VAR
TEST('Check_DWORD_TO_WORD_TooHigh');

// @TEST-RUN
converted := TryConvert_DWORD_TO_Destination(value, actual);

// @TEST-ASSERT
AssertFalse(Condition := converted, Message := 'Did not report DWORD to WORD conversion was prevented');

TEST_FINISHED();
END_METHOD

END_FUNCTION_BLOCK

// ---- mobject-converters/Tests/SINT_TO_TestSuite.TcPOU
FUNCTION_BLOCK PUBLIC SINT_TO_TestSuite EXTENDS TcUnit.FB_TestSuite
VAR
END_VAR

Check_SINT_TO_BOOL_Max();
Check_SINT_TO_BOOL_Min();
Check_SINT_TO_BYTE_Max();
Check_SINT_TO_BYTE_Min();
Check_SINT_TO_BYTE_TooLow();
Check_SINT_TO_WORD_Max();
Check_SINT_TO_WORD_Min();
Check_SINT_TO_WORD_TooLow();
Check_SINT_TO_DWORD_Max();
Check_SINT_TO_DWORD_Min();
Check_SINT_TO_DWORD_TooLow();
Check_SINT_TO_LWORD_Max();
Check_SINT_TO_LWORD_Min();
Check_SINT_TO_LWORD_TooLow();
Check_SINT_TO_SINT_Max();
Check_SINT_TO_SINT_Min();
Check_SINT_TO_INT_Max();
Check_SINT_TO_INT_Min();
Check_SINT_TO_DINT_Max();
Check_SINT_TO_DINT_Min();
Check_SINT_TO_LINT_Max();
Check_SINT_TO_LINT_Min();
Check_SINT_TO_USINT_Max();
Check_SINT_TO_USINT_Min();
Check_SINT_TO_USINT_TooLow();
Check_SINT_TO_UINT_Max();
Check_SINT_TO_UINT_Min();
Check_SINT_TO_UINT_TooLow();
Check_SINT_TO_UDINT_Max();
Check_SINT_TO_UDINT_Min();
Check_SINT_TO_UDINT_TooLow();
Check_SINT_TO_ULINT_Max();
Check_SINT_TO_ULINT_Min();
Check_SINT_TO_ULINT_TooLow();
Check_SINT_TO_REAL_Max();
Check_SINT_TO_REAL_Min();
Check_SINT_TO_LREAL_Max();
Check_SINT_TO_LREAL_Min();
Check_SINT_TO_TIME_Max();
Check_SINT_TO_TIME_Min();
Check_SINT_TO_TIME_TooLow();
Check_SINT_TO_TOD_Max();
Check_SINT_TO_TOD_Min();
Check_SINT_TO_TOD_TooLow();
Check_SINT_TO_DATE_Max();
Check_SINT_TO_DATE_Min();
Check_SINT_TO_DATE_TooLow();
Check_SINT_TO_DT_Max();
Check_SINT_TO_DT_Min();
Check_SINT_TO_DT_TooLow();
Check_SINT_TO_STRING_Max();
Check_SINT_TO_STRING_Min();

METHOD PUBLIC Check_SINT_TO_BOOL_Max
VAR
	value : SINT := DatatypeLimits.SINT_MAX_VALUE;
	actual : BOOL;
	converted : BOOL;
	equal : BOOL;
END_VAR
TEST('Check_SINT_TO_BOOL_Max');

// @TEST-RUN
converted := TryConvert_SINT_TO_Destination(value, actual);
equal := actual = SINT_TO_BOOL(value);

// @TEST-ASSERT
AssertTrue(Condition := equal, Message := 'Did not convert SINT to BOOL correctly');
AssertTrue(Condition := converted, Message := 'Did not report SINT to BOOL conversion was successful');

TEST_FINISHED();
END_METHOD

METHOD PUBLIC Check_SINT_TO_BOOL_Min
VAR
	value : SINT := DatatypeLimits.SINT_MIN_VALUE;
	actual : BOOL;
	converted : BOOL;
	equal : BOOL;
END_VAR
TEST('Check_SINT_TO_BOOL_Min');

// @TEST-RUN
converted := TryConvert_SINT_TO_Destination(value, actual);
equal := actual = SINT_TO_BOOL(value);

// @TEST-ASSERT
AssertTrue(Condition := equal, Message := 'Did not convert SINT to BOOL correctly');
AssertTrue(Condition := converted, Message := 'Did not report SINT to BOOL conversion was successful');

TEST_FINISHED();
END_METHOD

METHOD PUBLIC Check_SINT_TO_BYTE_Max
VAR
	value : SINT := DatatypeLimits.SINT_MAX_VALUE;
	actual : BYTE;
	converted : BOOL;
	equal : BOOL;
END_VAR
TEST('Check_SINT_TO_BYTE_Max');

// @TEST-RUN
converted := TryConvert_SINT_TO_Destination(value, actual);
equal := actual = SINT_TO_BYTE(value);

// @TEST-ASSERT
AssertTrue(Condition := equal, Message := 'Did not convert SINT to BYTE correctly');
AssertTrue(Condition := converted, Message := 'Did not report SINT to BYTE conversion was successful');

TEST_FINISHED();
END_METHOD

METHOD PUBLIC Check_SINT_TO_BYTE_Min
VAR
	value : SINT := DatatypeLimits.MIN_VALUE_OF_SINT_WHICH_CAN_BE_HELD_IN_A_BYTE;
	actual : BYTE;
	converted : BOOL;
	equal : BOOL;
END_VAR
TEST('Check_SINT_TO_BYTE_Min');

// @TEST-RUN
converted := TryConvert_SINT_TO_Destination(value, actual);
equal := actual = SINT_TO_BYTE(value);

// @TEST-ASSERT
AssertTrue(Condition := equal, Message := 'Did not convert SINT to BYTE correctly');
AssertTrue(Condition := converted, Message := 'Did not report SINT to BYTE conversion was successful');

TEST_FINISHED();
END_METHOD

METHOD PUBLIC Check_SINT_TO_BYTE_TooLow
VAR
	value : SINT := DatatypeLimits.SINT_MIN_VALUE;
	actual : BYTE;
	converted : BOOL;
END_VAR
TEST('Check_SINT_TO_BYTE_TooLow');

// @TEST-RUN
converted := TryConvert_SINT_TO_Destination(value, actual);

// @TEST-ASSERT
AssertFalse(Condition := converted, Message := 'Did not report SINT to BYTE conversion was prevented');

TEST_FINISHED();
END_METHOD

METHOD PUBLIC Check_SINT_TO_DATE_Max
VAR
	value : SINT := DatatypeLimits.SINT_MAX_VALUE;
	actual : DATE;
	converted : BOOL;
	equal : BOOL;
END_VAR
TEST('Check_SINT_TO_DATE_Max');

// @TEST-RUN
converted := TryConvert_SINT_TO_Destination(value, actual);
equal := actual = SINT_TO_DATE(value);

// @TEST-ASSERT
AssertTrue(Condition := equal, Message := 'Did not convert SINT to DATE correctly');
AssertTrue(Condition := converted, Message := 'Did not report SINT to DATE conversion was successful');

TEST_FINISHED();
END_METHOD

METHOD PUBLIC Check_SINT_TO_DATE_Min
VAR
	value : SINT := DatatypeLimits.MIN_VALUE_OF_SINT_WHICH_CAN_BE_HELD_IN_A_DATE;
	actual : DATE;
	converted : BOOL;
	equal : BOOL;
END_VAR
TEST('Check_SINT_TO_DATE_Min');

// @TEST-RUN
converted := TryConvert_SINT_TO_Destination(value, actual);
equal := actual = SINT_TO_DATE(value);

// @TEST-ASSERT
AssertTrue(Condition := equal, Message := 'Did not convert SINT to DATE correctly');
AssertTrue(Condition := converted, Message := 'Did not report SINT to DATE conversion was successful');

TEST_FINISHED();
END_METHOD

METHOD PUBLIC Check_SINT_TO_DATE_TooLow
VAR
	value : SINT := DatatypeLimits.SINT_MIN_VALUE;
	actual : DATE;
	converted : BOOL;
END_VAR
TEST('Check_SINT_TO_DATE_TooLow');

// @TEST-RUN
converted := TryConvert_SINT_TO_Destination(value, actual);

// @TEST-ASSERT
AssertFalse(Condition := converted, Message := 'Did not report SINT to DATE conversion was prevented');

TEST_FINISHED();
END_METHOD

METHOD PUBLIC Check_SINT_TO_DINT_Max
VAR
	value : SINT := DatatypeLimits.SINT_MAX_VALUE;
	actual : DINT;
	converted : BOOL;
	equal : BOOL;
END_VAR
TEST('Check_SINT_TO_DINT_Max');

// @TEST-RUN
converted := TryConvert_SINT_TO_Destination(value, actual);
equal := actual = SINT_TO_DINT(value);

// @TEST-ASSERT
AssertTrue(Condition := equal, Message := 'Did not convert SINT to DINT correctly');
AssertTrue(Condition := converted, Message := 'Did not report SINT to DINT conversion was successful');

TEST_FINISHED();
END_METHOD

METHOD PUBLIC Check_SINT_TO_DINT_Min
VAR
	value : SINT := DatatypeLimits.SINT_MIN_VALUE;
	actual : DINT;
	converted : BOOL;
	equal : BOOL;
END_VAR
TEST('Check_SINT_TO_DINT_Min');

// @TEST-RUN
converted := TryConvert_SINT_TO_Destination(value, actual);
equal := actual = SINT_TO_DINT(value);

// @TEST-ASSERT
AssertTrue(Condition := equal, Message := 'Did not convert SINT to DINT correctly');
AssertTrue(Condition := converted, Message := 'Did not report SINT to DINT conversion was successful');

TEST_FINISHED();
END_METHOD

METHOD PUBLIC Check_SINT_TO_DT_Max
VAR
	value : SINT := DatatypeLimits.SINT_MAX_VALUE;
	actual : DT;
	converted : BOOL;
	equal : BOOL;
END_VAR
TEST('Check_SINT_TO_DT_Max');

// @TEST-RUN
converted := TryConvert_SINT_TO_Destination(value, actual);
equal := actual = SINT_TO_DT(value);

// @TEST-ASSERT
AssertTrue(Condition := equal, Message := 'Did not convert SINT to DT correctly');
AssertTrue(Condition := converted, Message := 'Did not report SINT to DT conversion was successful');

TEST_FINISHED();
END_METHOD

METHOD PUBLIC Check_SINT_TO_DT_Min
VAR
	value : SINT := DatatypeLimits.MIN_VALUE_OF_SINT_WHICH_CAN_BE_HELD_IN_A_DT;
	actual : DT;
	converted : BOOL;
	equal : BOOL;
END_VAR
TEST('Check_SINT_TO_DT_Min');

// @TEST-RUN
converted := TryConvert_SINT_TO_Destination(value, actual);
equal := actual = SINT_TO_DT(value);

// @TEST-ASSERT
AssertTrue(Condition := equal, Message := 'Did not convert SINT to DT correctly');
AssertTrue(Condition := converted, Message := 'Did not report SINT to DT conversion was successful');

TEST_FINISHED();
END_METHOD

METHOD PUBLIC Check_SINT_TO_DT_TooLow
VAR
	value : SINT := DatatypeLimits.SINT_MIN_VALUE;
	actual : DT;
	converted : BOOL;
END_VAR
TEST('Check_SINT_TO_DT_TooLow');

// @TEST-RUN
converted := TryConvert_SINT_TO_Destination(value, actual);

// @TEST-ASSERT
AssertFalse(Condition := converted, Message := 'Did not report SINT to DT conversion was prevented');

TEST_FINISHED();
END_METHOD

METHOD PUBLIC Check_SINT_TO_DWORD_Max
VAR
	value : SINT := DatatypeLimits.SINT_MAX_VALUE;
	actual : DWORD;
	converted : BOOL;
	equal : BOOL;
END_VAR
TEST('Check_SINT_TO_DWORD_Max');

// @TEST-RUN
converted := TryConvert_SINT_TO_Destination(value, actual);
equal := actual = SINT_TO_DWORD(value);

// @TEST-ASSERT
AssertTrue(Condition := equal, Message := 'Did not convert SINT to DWORD correctly');
AssertTrue(Condition := converted, Message := 'Did not report SINT to DWORD conversion was successful');

TEST_FINISHED();
END_METHOD

METHOD PUBLIC Check_SINT_TO_DWORD_Min
VAR
	value : SINT := DatatypeLimits.MIN_VALUE_OF_SINT_WHICH_CAN_BE_HELD_IN_A_DWORD;
	actual : DWORD;
	converted : BOOL;
	equal : BOOL;
END_VAR
TEST('Check_SINT_TO_DWORD_Min');

// @TEST-RUN
converted := TryConvert_SINT_TO_Destination(value, actual);
equal := actual = SINT_TO_DWORD(value);

// @TEST-ASSERT
AssertTrue(Condition := equal, Message := 'Did not convert SINT to DWORD correctly');
AssertTrue(Condition := converted, Message := 'Did not report SINT to DWORD conversion was successful');

TEST_FINISHED();
END_METHOD

METHOD PUBLIC Check_SINT_TO_DWORD_TooLow
VAR
	value : SINT := DatatypeLimits.SINT_MIN_VALUE;
	actual : DWORD;
	converted : BOOL;
END_VAR
TEST('Check_SINT_TO_DWORD_TooLow');

// @TEST-RUN
converted := TryConvert_SINT_TO_Destination(value, actual);

// @TEST-ASSERT
AssertFalse(Condition := converted, Message := 'Did not report SINT to DWORD conversion was prevented');

TEST_FINISHED();
END_METHOD

METHOD PUBLIC Check_SINT_TO_INT_Max
VAR
	value : SINT := DatatypeLimits.SINT_MAX_VALUE;
	actual : INT;
	converted : BOOL;
	equal : BOOL;
END_VAR
TEST('Check_SINT_TO_INT_Max');

// @TEST-RUN
converted := TryConvert_SINT_TO_Destination(value, actual);
equal := actual = SINT_TO_INT(value);

// @TEST-ASSERT
AssertTrue(Condition := equal, Message := 'Did not convert SINT to INT correctly');
AssertTrue(Condition := converted, Message := 'Did not report SINT to INT conversion was successful');

TEST_FINISHED();
END_METHOD

METHOD PUBLIC Check_SINT_TO_INT_Min
VAR
	value : SINT := DatatypeLimits.SINT_MIN_VALUE;
	actual : INT;
	converted : BOOL;
	equal : BOOL;
END_VAR
TEST('Check_SINT_TO_INT_Min');

// @TEST-RUN
converted := TryConvert_SINT_TO_Destination(value, actual);
equal := actual = SINT_TO_INT(value);

// @TEST-ASSERT
AssertTrue(Condition := equal, Message := 'Did not convert SINT to INT correctly');
AssertTrue(Condition := converted, Message := 'Did not report SINT to INT conversion was successful');

TEST_FINISHED();
END_METHOD

METHOD PUBLIC Check_SINT_TO_LINT_Max
VAR
	value : SINT := DatatypeLimits.SINT_MAX_VALUE;
	actual : LINT;
	converted : BOOL;
	equal : BOOL;
END_VAR
TEST('Check_SINT_TO_LINT_Max');

// @TEST-RUN
converted := TryConvert_SINT_TO_Destination(value, actual);
equal := actual = SINT_TO_LINT(value);

// @TEST-ASSERT
AssertTrue(Condition := equal, Message := 'Did not convert SINT to LINT correctly');
AssertTrue(Condition := converted, Message := 'Did not report SINT to LINT conversion was successful');

TEST_FINISHED();
END_METHOD

METHOD PUBLIC Check_SINT_TO_LINT_Min
VAR
	value : SINT := DatatypeLimits.SINT_MIN_VALUE;
	actual : LINT;
	converted : BOOL;
	equal : BOOL;
END_VAR
TEST('Check_SINT_TO_LINT_Min');

// @TEST-RUN
converted := TryConvert_SINT_TO_Destination(value, actual);
equal := actual = SINT_TO_LINT(value);

// @TEST-ASSERT
AssertTrue(Condition := equal, Message := 'Did not convert SINT to LINT correctly');
AssertTrue(Condition := converted, Message := 'Did not report SINT to LINT conversion was successful');

TEST_FINISHED();
END_METHOD

METHOD PUBLIC Check_SINT_TO_LREAL_Max
VAR
	value : SINT := DatatypeLimits.SINT_MAX_VALUE;
	actual : LREAL;
	converted : BOOL;
	equal : BOOL;
END_VAR
TEST('Check_SINT_TO_LREAL_Max');

// @TEST-RUN
converted := TryConvert_SINT_TO_Destination(value, actual);
equal := actual = SINT_TO_LREAL(value);

// @TEST-ASSERT
AssertTrue(Condition := equal, Message := 'Did not convert SINT to LREAL correctly');
AssertTrue(Condition := converted, Message := 'Did not report SINT to LREAL conversion was successful');

TEST_FINISHED();
END_METHOD

METHOD PUBLIC Check_SINT_TO_LREAL_Min
VAR
	value : SINT := DatatypeLimits.SINT_MIN_VALUE;
	actual : LREAL;
	converted : BOOL;
	equal : BOOL;
END_VAR
TEST('Check_SINT_TO_LREAL_Min');

// @TEST-RUN
converted := TryConvert_SINT_TO_Destination(value, actual);
equal := actual = SINT_TO_LREAL(value);

// @TEST-ASSERT
AssertTrue(Condition := equal, Message := 'Did not convert SINT to LREAL correctly');
AssertTrue(Condition := converted, Message := 'Did not report SINT to LREAL conversion was successful');

TEST_FINISHED();
END_METHOD

METHOD PUBLIC Check_SINT_TO_LWORD_Max
VAR
	value : SINT := DatatypeLimits.SINT_MAX_VALUE;
	actual : LWORD;
	converted : BOOL;
	equal : BOOL;
END_VAR
TEST('Check_SINT_TO_LWORD_Max');

// @TEST-RUN
converted := TryConvert_SINT_TO_Destination(value, actual);
equal := actual = SINT_TO_LWORD(value);

// @TEST-ASSERT
AssertTrue(Condition := equal, Message := 'Did not convert SINT to LWORD correctly');
AssertTrue(Condition := converted, Message := 'Did not report SINT to LWORD conversion was successful');

TEST_FINISHED();
END_METHOD

METHOD PUBLIC Check_SINT_TO_LWORD_Min
VAR
	value : SINT := DatatypeLimits.MIN_VALUE_OF_SINT_WHICH_CAN_BE_HELD_IN_A_LWORD;
	actual : LWORD;
	converted : BOOL;
	equal : BOOL;
END_VAR
TEST('Check_SINT_TO_LWORD_Min');

// @TEST-RUN
converted := TryConvert_SINT_TO_Destination(value, actual);
equal := actual = SINT_TO_LWORD(value);

// @TEST-ASSERT
AssertTrue(Condition := equal, Message := 'Did not convert SINT to LWORD correctly');
AssertTrue(Condition := converted, Message := 'Did not report SINT to LWORD conversion was successful');

TEST_FINISHED();
END_METHOD

METHOD PUBLIC Check_SINT_TO_LWORD_TooLow
VAR
	value : SINT := DatatypeLimits.SINT_MIN_VALUE;
	actual : LWORD;
	converted : BOOL;
END_VAR
TEST('Check_SINT_TO_LWORD_TooLow');

// @TEST-RUN
converted := TryConvert_SINT_TO_Destination(value, actual);

// @TEST-ASSERT
AssertFalse(Condition := converted, Message := 'Did not report SINT to LWORD conversion was prevented');

TEST_FINISHED();
END_METHOD

METHOD PUBLIC Check_SINT_TO_REAL_Max
VAR
	value : SINT := DatatypeLimits.SINT_MAX_VALUE;
	actual : REAL;
	converted : BOOL;
	equal : BOOL;
END_VAR
TEST('Check_SINT_TO_REAL_Max');

// @TEST-RUN
converted := TryConvert_SINT_TO_Destination(value, actual);
equal := actual = SINT_TO_REAL(value);

// @TEST-ASSERT
AssertTrue(Condition := equal, Message := 'Did not convert SINT to REAL correctly');
AssertTrue(Condition := converted, Message := 'Did not report SINT to REAL conversion was successful');

TEST_FINISHED();
END_METHOD

METHOD PUBLIC Check_SINT_TO_REAL_Min
VAR
	value : SINT := DatatypeLimits.SINT_MIN_VALUE;
	actual : REAL;
	converted : BOOL;
	equal : BOOL;
END_VAR
TEST('Check_SINT_TO_REAL_Min');

// @TEST-RUN
converted := TryConvert_SINT_TO_Destination(value, actual);
equal := actual = SINT_TO_REAL(value);

// @TEST-ASSERT
AssertTrue(Condition := equal, Message := 'Did not convert SINT to REAL correctly');
AssertTrue(Condition := converted, Message := 'Did not report SINT to REAL conversion was successful');

TEST_FINISHED();
END_METHOD

METHOD PUBLIC Check_SINT_TO_SINT_Max
VAR
	value : SINT := DatatypeLimits.SINT_MAX_VALUE;
	actual : SINT;
	converted : BOOL;
	equal : BOOL;
END_VAR
TEST('Check_SINT_TO_SINT_Max');

// @TEST-RUN
converted := TryConvert_SINT_TO_Destination(value, actual);
equal := actual = value;

// @TEST-ASSERT
AssertTrue(Condition := equal, Message := 'Did not convert SINT to SINT correctly');
AssertTrue(Condition := converted, Message := 'Did not report SINT to SINT conversion was successful');

TEST_FINISHED();
END_METHOD

METHOD PUBLIC Check_SINT_TO_SINT_Min
VAR
	value : SINT := DatatypeLimits.SINT_MIN_VALUE;
	actual : SINT;
	converted : BOOL;
	equal : BOOL;
END_VAR
TEST('Check_SINT_TO_SINT_Min');

// @TEST-RUN
converted := TryConvert_SINT_TO_Destination(value, actual);
equal := actual = value;

// @TEST-ASSERT
AssertTrue(Condition := equal, Message := 'Did not convert SINT to SINT correctly');
AssertTrue(Condition := converted, Message := 'Did not report SINT to SINT conversion was successful');

TEST_FINISHED();
END_METHOD

METHOD PUBLIC Check_SINT_TO_STRING_Max
VAR
	value : SINT := DatatypeLimits.SINT_MAX_VALUE;
	actual : STRING;
	converted : BOOL;
	equal : BOOL;
END_VAR
TEST('Check_SINT_TO_STRING_Max');

// @TEST-RUN
converted := TryConvert_SINT_TO_Destination(value, actual);
equal := actual = SINT_TO_STRING(value);

// @TEST-ASSERT
AssertTrue(Condition := equal, Message := 'Did not convert SINT to STRING correctly');
AssertTrue(Condition := converted, Message := 'Did not report SINT to STRING conversion was successful');

TEST_FINISHED();
END_METHOD

METHOD PUBLIC Check_SINT_TO_STRING_Min
VAR
	value : SINT := DatatypeLimits.SINT_MIN_VALUE;
	actual : STRING;
	converted : BOOL;
	equal : BOOL;
END_VAR
TEST('Check_SINT_TO_STRING_Min');

// @TEST-RUN
converted := TryConvert_SINT_TO_Destination(value, actual);
equal := actual = SINT_TO_STRING(value);

// @TEST-ASSERT
AssertTrue(Condition := equal, Message := 'Did not convert SINT to STRING correctly');
AssertTrue(Condition := converted, Message := 'Did not report SINT to STRING conversion was successful');

TEST_FINISHED();
END_METHOD

METHOD PUBLIC Check_SINT_TO_TIME_Max
VAR
	value : SINT := DatatypeLimits.SINT_MAX_VALUE;
	actual : TIME;
	converted : BOOL;
	equal : BOOL;
END_VAR
TEST('Check_SINT_TO_TIME_Max');

// @TEST-RUN
converted := TryConvert_SINT_TO_Destination(value, actual);
equal := actual = SINT_TO_TIME(value);

// @TEST-ASSERT
AssertTrue(Condition := equal, Message := 'Did not convert SINT to TIME correctly');
AssertTrue(Condition := converted, Message := 'Did not report SINT to TIME conversion was successful');

TEST_FINISHED();
END_METHOD

METHOD PUBLIC Check_SINT_TO_TIME_Min
VAR
	value : SINT := DatatypeLimits.MIN_VALUE_OF_SINT_WHICH_CAN_BE_HELD_IN_A_TIME;
	actual : TIME;
	converted : BOOL;
	equal : BOOL;
END_VAR
TEST('Check_SINT_TO_TIME_Min');

// @TEST-RUN
converted := TryConvert_SINT_TO_Destination(value, actual);
equal := actual = SINT_TO_TIME(value);

// @TEST-ASSERT
AssertTrue(Condition := equal, Message := 'Did not convert SINT to TIME correctly');
AssertTrue(Condition := converted, Message := 'Did not report SINT to TIME conversion was successful');

TEST_FINISHED();
END_METHOD

METHOD PUBLIC Check_SINT_TO_TIME_TooLow
VAR
	value : SINT := DatatypeLimits.SINT_MIN_VALUE;
	actual : TIME;
	converted : BOOL;
END_VAR
TEST('Check_SINT_TO_TIME_TooLow');

// @TEST-RUN
converted := TryConvert_SINT_TO_Destination(value, actual);

// @TEST-ASSERT
AssertFalse(Condition := converted, Message := 'Did not report SINT to TIME conversion was prevented');

TEST_FINISHED();
END_METHOD

METHOD PUBLIC Check_SINT_TO_TOD_Max
VAR
	value : SINT := DatatypeLimits.SINT_MAX_VALUE;
	actual : TOD;
	converted : BOOL;
	equal : BOOL;
END_VAR
TEST('Check_SINT_TO_TOD_Max');

// @TEST-RUN
converted := TryConvert_SINT_TO_Destination(value, actual);
equal := actual = SINT_TO_TOD(value);

// @TEST-ASSERT
AssertTrue(Condition := equal, Message := 'Did not convert SINT to TOD correctly');
AssertTrue(Condition := converted, Message := 'Did not report SINT to TOD conversion was successful');

TEST_FINISHED();
END_METHOD

METHOD PUBLIC Check_SINT_TO_TOD_Min
VAR
	value : SINT := DatatypeLimits.MIN_VALUE_OF_SINT_WHICH_CAN_BE_HELD_IN_A_TOD;
	actual : TOD;
	converted : BOOL;
	equal : BOOL;
END_VAR
TEST('Check_SINT_TO_TOD_Min');

// @TEST-RUN
converted := TryConvert_SINT_TO_Destination(value, actual);
equal := actual = SINT_TO_TOD(value);

// @TEST-ASSERT
AssertTrue(Condition := equal, Message := 'Did not convert SINT to TOD correctly');
AssertTrue(Condition := converted, Message := 'Did not report SINT to TOD conversion was successful');

TEST_FINISHED();
END_METHOD

METHOD PUBLIC Check_SINT_TO_TOD_TooLow
VAR
	value : SINT := DatatypeLimits.SINT_MIN_VALUE;
	actual : TOD;
	converted : BOOL;
END_VAR
TEST('Check_SINT_TO_TOD_TooLow');

// @TEST-RUN
converted := TryConvert_SINT_TO_Destination(value, actual);

// @TEST-ASSERT
AssertFalse(Condition := converted, Message := 'Did not report SINT to TOD conversion was prevented');

TEST_FINISHED();
END_METHOD

METHOD PUBLIC Check_SINT_TO_UDINT_Max
VAR
	value : SINT := DatatypeLimits.SINT_MAX_VALUE;
	actual : UDINT;
	converted : BOOL;
	equal : BOOL;
END_VAR
TEST('Check_SINT_TO_UDINT_Max');

// @TEST-RUN
converted := TryConvert_SINT_TO_Destination(value, actual);
equal := actual = SINT_TO_UDINT(value);

// @TEST-ASSERT
AssertTrue(Condition := equal, Message := 'Did not convert SINT to UDINT correctly');
AssertTrue(Condition := converted, Message := 'Did not report SINT to UDINT conversion was successful');

TEST_FINISHED();
END_METHOD

METHOD PUBLIC Check_SINT_TO_UDINT_Min
VAR
	value : SINT := DatatypeLimits.MIN_VALUE_OF_SINT_WHICH_CAN_BE_HELD_IN_A_UDINT;
	actual : UDINT;
	converted : BOOL;
	equal : BOOL;
END_VAR
TEST('Check_SINT_TO_UDINT_Min');

// @TEST-RUN
converted := TryConvert_SINT_TO_Destination(value, actual);
equal := actual = SINT_TO_UDINT(value);

// @TEST-ASSERT
AssertTrue(Condition := equal, Message := 'Did not convert SINT to UDINT correctly');
AssertTrue(Condition := converted, Message := 'Did not report SINT to UDINT conversion was successful');

TEST_FINISHED();
END_METHOD

METHOD PUBLIC Check_SINT_TO_UDINT_TooLow
VAR
	value : SINT := DatatypeLimits.SINT_MIN_VALUE;
	actual : UDINT;
	converted : BOOL;
END_VAR
TEST('Check_SINT_TO_UDINT_TooLow');

// @TEST-RUN
converted := TryConvert_SINT_TO_Destination(value, actual);

// @TEST-ASSERT
AssertFalse(Condition := converted, Message := 'Did not report SINT to UDINT conversion was prevented');

TEST_FINISHED();
END_METHOD

METHOD PUBLIC Check_SINT_TO_UINT_Max
VAR
	value : SINT := DatatypeLimits.SINT_MAX_VALUE;
	actual : UINT;
	converted : BOOL;
	equal : BOOL;
END_VAR
TEST('Check_SINT_TO_UINT_Max');

// @TEST-RUN
converted := TryConvert_SINT_TO_Destination(value, actual);
equal := actual = SINT_TO_UINT(value);

// @TEST-ASSERT
AssertTrue(Condition := equal, Message := 'Did not convert SINT to UINT correctly');
AssertTrue(Condition := converted, Message := 'Did not report SINT to UINT conversion was successful');

TEST_FINISHED();
END_METHOD

METHOD PUBLIC Check_SINT_TO_UINT_Min
VAR
	value : SINT := DatatypeLimits.MIN_VALUE_OF_SINT_WHICH_CAN_BE_HELD_IN_A_UINT;
	actual : UINT;
	converted : BOOL;
	equal : BOOL;
END_VAR
TEST('Check_SINT_TO_UINT_Min');

// @TEST-RUN
converted := TryConvert_SINT_TO_Destination(value, actual);
equal := actual = SINT_TO_UINT(value);

// @TEST-ASSERT
AssertTrue(Condition := equal, Message := 'Did not convert SINT to UINT correctly');
AssertTrue(Condition := converted, Message := 'Did not report SINT to UINT conversion was successful');

TEST_FINISHED();
END_METHOD

METHOD PUBLIC Check_SINT_TO_UINT_TooLow
VAR
	value : SINT := DatatypeLimits.SINT_MIN_VALUE;
	actual : UINT;
	converted : BOOL;
END_VAR
TEST('Check_SINT_TO_UINT_TooLow');

// @TEST-RUN
converted := TryConvert_SINT_TO_Destination(value, actual);

// @TEST-ASSERT
AssertFalse(Condition := converted, Message := 'Did not report SINT to UINT conversion was prevented');

TEST_FINISHED();
END_METHOD

METHOD PUBLIC Check_SINT_TO_ULINT_Max
VAR
	value : SINT := DatatypeLimits.SINT_MAX_VALUE;
	actual : ULINT;
	converted : BOOL;
	equal : BOOL;
END_VAR
TEST('Check_SINT_TO_ULINT_Max');

// @TEST-RUN
converted := TryConvert_SINT_TO_Destination(value, actual);
equal := actual = SINT_TO_ULINT(value);

// @TEST-ASSERT
AssertTrue(Condition := equal, Message := 'Did not convert SINT to ULINT correctly');
AssertTrue(Condition := converted, Message := 'Did not report SINT to ULINT conversion was successful');

TEST_FINISHED();
END_METHOD

METHOD PUBLIC Check_SINT_TO_ULINT_Min
VAR
	value : SINT := DatatypeLimits.MIN_VALUE_OF_SINT_WHICH_CAN_BE_HELD_IN_A_ULINT;
	actual : ULINT;
	converted : BOOL;
	equal : BOOL;
END_VAR
TEST('Check_SINT_TO_ULINT_Min');

// @TEST-RUN
converted := TryConvert_SINT_TO_Destination(value, actual);
equal := actual = SINT_TO_ULINT(value);

// @TEST-ASSERT
AssertTrue(Condition := equal, Message := 'Did not convert SINT to ULINT correctly');
AssertTrue(Condition := converted, Message := 'Did not report SINT to ULINT conversion was successful');

TEST_FINISHED();
END_METHOD

METHOD PUBLIC Check_SINT_TO_ULINT_TooLow
VAR
	value : SINT := DatatypeLimits.SINT_MIN_VALUE;
	actual : ULINT;
	converted : BOOL;
END_VAR
TEST('Check_SINT_TO_ULINT_TooLow');

// @TEST-RUN
converted := TryConvert_SINT_TO_Destination(value, actual);

// @TEST-ASSERT
AssertFalse(Condition := converted, Message := 'Did not report SINT to ULINT conversion was prevented');

TEST_FINISHED();
END_METHOD

METHOD PUBLIC Check_SINT_TO_USINT_Max
VAR
	value : SINT := DatatypeLimits.SINT_MAX_VALUE;
	actual : USINT;
	converted : BOOL;
	equal : BOOL;
END_VAR
TEST('Check_SINT_TO_USINT_Max');

// @TEST-RUN
converted := TryConvert_SINT_TO_Destination(value, actual);
equal := actual = SINT_TO_USINT(value);

// @TEST-ASSERT
AssertTrue(Condition := equal, Message := 'Did not convert SINT to USINT correctly');
AssertTrue(Condition := converted, Message := 'Did not report SINT to USINT conversion was successful');

TEST_FINISHED();
END_METHOD

METHOD PUBLIC Check_SINT_TO_USINT_Min
VAR
	value : SINT := DatatypeLimits.MIN_VALUE_OF_SINT_WHICH_CAN_BE_HELD_IN_A_USINT;
	actual : USINT;
	converted : BOOL;
	equal : BOOL;
END_VAR
TEST('Check_SINT_TO_USINT_Min');

// @TEST-RUN
converted := TryConvert_SINT_TO_Destination(value, actual);
equal := actual = SINT_TO_USINT(value);

// @TEST-ASSERT
AssertTrue(Condition := equal, Message := 'Did not convert SINT to USINT correctly');
AssertTrue(Condition := converted, Message := 'Did not report SINT to USINT conversion was successful');

TEST_FINISHED();
END_METHOD

METHOD PUBLIC Check_SINT_TO_USINT_TooLow
VAR
	value : SINT := DatatypeLimits.SINT_MIN_VALUE;
	actual : USINT;
	converted : BOOL;
END_VAR
TEST('Check_SINT_TO_USINT_TooLow');

// @TEST-RUN
converted := TryConvert_SINT_TO_Destination(value, actual);

// @TEST-ASSERT
AssertFalse(Condition := converted, Message := 'Did not report SINT to USINT conversion was prevented');

TEST_FINISHED();
END_METHOD

METHOD PUBLIC Check_SINT_TO_WORD_Max
VAR
	value : SINT := DatatypeLimits.SINT_MAX_VALUE;
	actual : WORD;
	converted : BOOL;
	equal : BOOL;
END_VAR
TEST('Check_SINT_TO_WORD_Max');

// @TEST-RUN
converted := TryConvert_SINT_TO_Destination(value, actual);
equal := actual = SINT_TO_WORD(value);

// @TEST-ASSERT
AssertTrue(Condition := equal, Message := 'Did not convert SINT to WORD correctly');
AssertTrue(Condition := converted, Message := 'Did not report SINT to WORD conversion was successful');

TEST_FINISHED();
END_METHOD

METHOD PUBLIC Check_SINT_TO_WORD_Min
VAR
	value : SINT := DatatypeLimits.MIN_VALUE_OF_SINT_WHICH_CAN_BE_HELD_IN_A_WORD;
	actual : WORD;
	converted : BOOL;
	equal : BOOL;
END_VAR
TEST('Check_SINT_TO_WORD_Min');

// @TEST-RUN
converted := TryConvert_SINT_TO_Destination(value, actual);
equal := actual = SINT_TO_WORD(value);

// @TEST-ASSERT
AssertTrue(Condition := equal, Message := 'Did not convert SINT to WORD correctly');
AssertTrue(Condition := converted, Message := 'Did not report SINT to WORD conversion was successful');

TEST_FINISHED();
END_METHOD

METHOD PUBLIC Check_SINT_TO_WORD_TooLow
VAR
	value : SINT := DatatypeLimits.SINT_MIN_VALUE;
	actual : WORD;
	converted : BOOL;
END_VAR
TEST('Check_SINT_TO_WORD_TooLow');

// @TEST-RUN
converted := TryConvert_SINT_TO_Destination(value, actual);

// @TEST-ASSERT
AssertFalse(Condition := converted, Message := 'Did not report SINT to WORD conversion was prevented');

TEST_FINISHED();
END_METHOD

END_FUNCTION_BLOCK

// ---- mobject-converters/Tests/UINT_TO_TestSuite.TcPOU
FUNCTION_BLOCK PUBLIC UINT_TO_TestSuite EXTENDS TcUnit.FB_TestSuite
VAR
END_VAR

Check_UINT_TO_BOOL_Max();
Check_UINT_TO_BOOL_Min();
Check_UINT_TO_BYTE_Max();
Check_UINT_TO_BYTE_Min();
Check_UINT_TO_BYTE_TooHigh();
Check_UINT_TO_WORD_Max();
Check_UINT_TO_WORD_Min();
Check_UINT_TO_DWORD_Max();
Check_UINT_TO_DWORD_Min();
Check_UINT_TO_LWORD_Max();
Check_UINT_TO_LWORD_Min();
Check_UINT_TO_SINT_Max();
Check_UINT_TO_SINT_Min();
Check_UINT_TO_SINT_TooHigh();
Check_UINT_TO_INT_Max();
Check_UINT_TO_INT_Min();
Check_UINT_TO_INT_TooHigh();
Check_UINT_TO_DINT_Max();
Check_UINT_TO_DINT_Min();
Check_UINT_TO_LINT_Max();
Check_UINT_TO_LINT_Min();
Check_UINT_TO_USINT_Max();
Check_UINT_TO_USINT_Min();
Check_UINT_TO_USINT_TooHigh();
Check_UINT_TO_UINT_Max();
Check_UINT_TO_UINT_Min();
Check_UINT_TO_UDINT_Max();
Check_UINT_TO_UDINT_Min();
Check_UINT_TO_ULINT_Max();
Check_UINT_TO_ULINT_Min();
Check_UINT_TO_REAL_Max();
Check_UINT_TO_REAL_Min();
Check_UINT_TO_LREAL_Max();
Check_UINT_TO_LREAL_Min();
Check_UINT_TO_TIME_Max();
Check_UINT_TO_TIME_Min();
Check_UINT_TO_TOD_Max();
Check_UINT_TO_TOD_Min();
Check_UINT_TO_DATE_Max();
Check_UINT_TO_DATE_Min();
Check_UINT_TO_DT_Max();
Check_UINT_TO_DT_Min();
Check_UINT_TO_STRING_Max();
Check_UINT_TO_STRING_Min();

METHOD PUBLIC Check_UINT_TO_BOOL_Max
VAR
	value : UINT := DatatypeLimits.UINT_MAX_VALUE;
	actual : BOOL;
	converted : BOOL;
	equal : BOOL;
END_VAR
TEST('Check_UINT_TO_BOOL_Max');

// @TEST-RUN
converted := TryConvert_UINT_TO_Destination(value, actual);
equal := actual = UINT_TO_BOOL(value);

// @TEST-ASSERT
AssertTrue(Condition := equal, Message := 'Did not convert UINT to BOOL correctly');
AssertTrue(Condition := converted, Message := 'Did not report UINT to BOOL conversion was successful');

TEST_FINISHED();
END_METHOD

METHOD PUBLIC Check_UINT_TO_BOOL_Min
VAR
	value : UINT := DatatypeLimits.UINT_MIN_VALUE;
	actual : BOOL;
	converted : BOOL;
	equal : BOOL;
END_VAR
TEST('Check_UINT_TO_BOOL_Min');

// @TEST-RUN
converted := TryConvert_UINT_TO_Destination(value, actual);
equal := actual = UINT_TO_BOOL(value);

// @TEST-ASSERT
AssertTrue(Condition := equal, Message := 'Did not convert UINT to BOOL correctly');
AssertTrue(Condition := converted, Message := 'Did not report UINT to BOOL conversion was successful');

TEST_FINISHED();
END_METHOD

METHOD PUBLIC Check_UINT_TO_BYTE_Max
VAR
	value : UINT := DatatypeLimits.MAX_VALUE_OF_UINT_WHICH_CAN_BE_HELD_IN_A_BYTE;
	actual : BYTE;
	converted : BOOL;
	equal : BOOL;
END_VAR
TEST('Check_UINT_TO_BYTE_Max');

// @TEST-RUN
converted := TryConvert_UINT_TO_Destination(value, actual);
equal := actual = UINT_TO_BYTE(value);

// @TEST-ASSERT
AssertTrue(Condition := equal, Message := 'Did not convert UINT to BYTE correctly');
AssertTrue(Condition := converted, Message := 'Did not report UINT to BYTE conversion was successful');

TEST_FINISHED();
END_METHOD

METHOD PUBLIC Check_UINT_TO_BYTE_Min
VAR
	value : UINT := DatatypeLimits.UINT_MIN_VALUE;
	actual : BYTE;
	converted : BOOL;
	equal : BOOL;
END_VAR
TEST('Check_UINT_TO_BYTE_Min');

// @TEST-RUN
converted := TryConvert_UINT_TO_Destination(value, actual);
equal := actual = UINT_TO_BYTE(value);

// @TEST-ASSERT
AssertTrue(Condition := equal, Message := 'Did not convert UINT to BYTE correctly');
AssertTrue(Condition := converted, Message := 'Did not report UINT to BYTE conversion was successful');

TEST_FINISHED();
END_METHOD

METHOD PUBLIC Check_UINT_TO_BYTE_TooHigh
VAR
	value : UINT := DatatypeLimits.UINT_MAX_VALUE;
	actual : BYTE;
	converted : BOOL;
END_VAR
TEST('Check_UINT_TO_BYTE_TooHigh');

// @TEST-RUN
converted := TryConvert_UINT_TO_Destination(value, actual);

// @TEST-ASSERT
AssertFalse(Condition := converted, Message := 'Did not report UINT to BYTE conversion was prevented');

TEST_FINISHED();
END_METHOD

METHOD PUBLIC Check_UINT_TO_DATE_Max
VAR
	value : UINT := DatatypeLimits.UINT_MAX_VALUE;
	actual : DATE;
	converted : BOOL;
	equal : BOOL;
END_VAR
TEST('Check_UINT_TO_DATE_Max');

// @TEST-RUN
converted := TryConvert_UINT_TO_Destination(value, actual);
equal := actual = UINT_TO_DATE(value);

// @TEST-ASSERT
AssertTrue(Condition := equal, Message := 'Did not convert UINT to DATE correctly');
AssertTrue(Condition := converted, Message := 'Did not report UINT to DATE conversion was successful');

TEST_FINISHED();
END_METHOD

METHOD PUBLIC Check_UINT_TO_DATE_Min
VAR
	value : UINT := DatatypeLimits.UINT_MIN_VALUE;
	actual : DATE;
	converted : BOOL;
	equal : BOOL;
END_VAR
TEST('Check_UINT_TO_DATE_Min');

// @TEST-RUN
converted := TryConvert_UINT_TO_Destination(value, actual);
equal := actual = UINT_TO_DATE(value);

// @TEST-ASSERT
AssertTrue(Condition := equal, Message := 'Did not convert UINT to DATE correctly');
AssertTrue(Condition := converted, Message := 'Did not report UINT to DATE conversion was successful');

TEST_FINISHED();
END_METHOD

METHOD PUBLIC Check_UINT_TO_DINT_Max
VAR
	value : UINT := DatatypeLimits.UINT_MAX_VALUE;
	actual : DINT;
	converted : BOOL;
	equal : BOOL;
END_VAR
TEST('Check_UINT_TO_DINT_Max');

// @TEST-RUN
converted := TryConvert_UINT_TO_Destination(value, actual);
equal := actual = UINT_TO_DINT(value);

// @TEST-ASSERT
AssertTrue(Condition := equal, Message := 'Did not convert UINT to DINT correctly');
AssertTrue(Condition := converted, Message := 'Did not report UINT to DINT conversion was successful');

TEST_FINISHED();
END_METHOD

METHOD PUBLIC Check_UINT_TO_DINT_Min
VAR
	value : UINT := DatatypeLimits.UINT_MIN_VALUE;
	actual : DINT;
	converted : BOOL;
	equal : BOOL;
END_VAR
TEST('Check_UINT_TO_DINT_Min');

// @TEST-RUN
converted := TryConvert_UINT_TO_Destination(value, actual);
equal := actual = UINT_TO_DINT(value);

// @TEST-ASSERT
AssertTrue(Condition := equal, Message := 'Did not convert UINT to DINT correctly');
AssertTrue(Condition := converted, Message := 'Did not report UINT to DINT conversion was successful');

TEST_FINISHED();
END_METHOD

METHOD PUBLIC Check_UINT_TO_DT_Max
VAR
	value : UINT := DatatypeLimits.UINT_MAX_VALUE;
	actual : DT;
	converted : BOOL;
	equal : BOOL;
END_VAR
TEST('Check_UINT_TO_DT_Max');

// @TEST-RUN
converted := TryConvert_UINT_TO_Destination(value, actual);
equal := actual = UINT_TO_DT(value);

// @TEST-ASSERT
AssertTrue(Condition := equal, Message := 'Did not convert UINT to DT correctly');
AssertTrue(Condition := converted, Message := 'Did not report UINT to DT conversion was successful');

TEST_FINISHED();
END_METHOD

METHOD PUBLIC Check_UINT_TO_DT_Min
VAR
	value : UINT := DatatypeLimits.UINT_MIN_VALUE;
	actual : DT;
	converted : BOOL;
	equal : BOOL;
END_VAR
TEST('Check_UINT_TO_DT_Min');

// @TEST-RUN
converted := TryConvert_UINT_TO_Destination(value, actual);
equal := actual = UINT_TO_DT(value);

// @TEST-ASSERT
AssertTrue(Condition := equal, Message := 'Did not convert UINT to DT correctly');
AssertTrue(Condition := converted, Message := 'Did not report UINT to DT conversion was successful');

TEST_FINISHED();
END_METHOD

METHOD PUBLIC Check_UINT_TO_DWORD_Max
VAR
	value : UINT := DatatypeLimits.UINT_MAX_VALUE;
	actual : DWORD;
	converted : BOOL;
	equal : BOOL;
END_VAR
TEST('Check_UINT_TO_DWORD_Max');

// @TEST-RUN
converted := TryConvert_UINT_TO_Destination(value, actual);
equal := actual = UINT_TO_DWORD(value);

// @TEST-ASSERT
AssertTrue(Condition := equal, Message := 'Did not convert UINT to DWORD correctly');
AssertTrue(Condition := converted, Message := 'Did not report UINT to DWORD conversion was successful');

TEST_FINISHED();
END_METHOD

METHOD PUBLIC Check_UINT_TO_DWORD_Min
VAR
	value : UINT := DatatypeLimits.UINT_MIN_VALUE;
	actual : DWORD;
	converted : BOOL;
	equal : BOOL;
END_VAR
TEST('Check_UINT_TO_DWORD_Min');

// @TEST-RUN
converted := TryConvert_UINT_TO_Destination(value, actual);
equal := actual = UINT_TO_DWORD(value);

// @TEST-ASSERT
AssertTrue(Condition := equal, Message := 'Did not convert UINT to DWORD correctly');
AssertTrue(Condition := converted, Message := 'Did not report UINT to DWORD conversion was successful');

TEST_FINISHED();
END_METHOD

METHOD PUBLIC Check_UINT_TO_INT_Max
VAR
	value : UINT := DatatypeLimits.MAX_VALUE_OF_UINT_WHICH_CAN_BE_HELD_IN_A_INT;
	actual : INT;
	converted : BOOL;
	equal : BOOL;
END_VAR
TEST('Check_UINT_TO_INT_Max');

// @TEST-RUN
converted := TryConvert_UINT_TO_Destination(value, actual);
equal := actual = UINT_TO_INT(value);

// @TEST-ASSERT
AssertTrue(Condition := equal, Message := 'Did not convert UINT to INT correctly');
AssertTrue(Condition := converted, Message := 'Did not report UINT to INT conversion was successful');

TEST_FINISHED();
END_METHOD

METHOD PUBLIC Check_UINT_TO_INT_Min
VAR
	value : UINT := DatatypeLimits.UINT_MIN_VALUE;
	actual : INT;
	converted : BOOL;
	equal : BOOL;
END_VAR
TEST('Check_UINT_TO_INT_Min');

// @TEST-RUN
converted := TryConvert_UINT_TO_Destination(value, actual);
equal := actual = UINT_TO_INT(value);

// @TEST-ASSERT
AssertTrue(Condition := equal, Message := 'Did not convert UINT to INT correctly');
AssertTrue(Condition := converted, Message := 'Did not report UINT to INT conversion was successful');

TEST_FINISHED();
END_METHOD

METHOD PUBLIC Check_UINT_TO_INT_TooHigh
VAR
	value : UINT := DatatypeLimits.UINT_MAX_VALUE;
	actual : INT;
	converted : BOOL;
END_VAR
TEST('Check_UINT_TO_INT_TooHigh');

// @TEST-RUN
converted := TryConvert_UINT_TO_Destination(value, actual);

// @TEST-ASSERT
AssertFalse(Condition := converted, Message := 'Did not report UINT to INT conversion was prevented');

TEST_FINISHED();
END_METHOD

METHOD PUBLIC Check_UINT_TO_LINT_Max
VAR
	value : UINT := DatatypeLimits.UINT_MAX_VALUE;
	actual : LINT;
	converted : BOOL;
	equal : BOOL;
END_VAR
TEST('Check_UINT_TO_LINT_Max');

// @TEST-RUN
converted := TryConvert_UINT_TO_Destination(value, actual);
equal := actual = UINT_TO_LINT(value);

// @TEST-ASSERT
AssertTrue(Condition := equal, Message := 'Did not convert UINT to LINT correctly');
AssertTrue(Condition := converted, Message := 'Did not report UINT to LINT conversion was successful');

TEST_FINISHED();
END_METHOD

METHOD PUBLIC Check_UINT_TO_LINT_Min
VAR
	value : UINT := DatatypeLimits.UINT_MIN_VALUE;
	actual : LINT;
	converted : BOOL;
	equal : BOOL;
END_VAR
TEST('Check_UINT_TO_LINT_Min');

// @TEST-RUN
converted := TryConvert_UINT_TO_Destination(value, actual);
equal := actual = UINT_TO_LINT(value);

// @TEST-ASSERT
AssertTrue(Condition := equal, Message := 'Did not convert UINT to LINT correctly');
AssertTrue(Condition := converted, Message := 'Did not report UINT to LINT conversion was successful');

TEST_FINISHED();
END_METHOD

METHOD PUBLIC Check_UINT_TO_LREAL_Max
VAR
	value : UINT := DatatypeLimits.UINT_MAX_VALUE;
	actual : LREAL;
	converted : BOOL;
	equal : BOOL;
END_VAR
TEST('Check_UINT_TO_LREAL_Max');

// @TEST-RUN
converted := TryConvert_UINT_TO_Destination(value, actual);
equal := actual = UINT_TO_LREAL(value);

// @TEST-ASSERT
AssertTrue(Condition := equal, Message := 'Did not convert UINT to LREAL correctly');
AssertTrue(Condition := converted, Message := 'Did not report UINT to LREAL conversion was successful');

TEST_FINISHED();
END_METHOD

METHOD PUBLIC Check_UINT_TO_LREAL_Min
VAR
	value : UINT := DatatypeLimits.UINT_MIN_VALUE;
	actual : LREAL;
	converted : BOOL;
	equal : BOOL;
END_VAR
TEST('Check_UINT_TO_LREAL_Min');

// @TEST-RUN
converted := TryConvert_UINT_TO_Destination(value, actual);
equal := actual = UINT_TO_LREAL(value);

// @TEST-ASSERT
AssertTrue(Condition := equal, Message := 'Did not convert UINT to LREAL correctly');
AssertTrue(Condition := converted, Message := 'Did not report UINT to LREAL conversion was successful');

TEST_FINISHED();
END_METHOD

METHOD PUBLIC Check_UINT_TO_LWORD_Max
VAR
	value : UINT := DatatypeLimits.UINT_MAX_VALUE;
	actual : LWORD;
	converted : BOOL;
	equal : BOOL;
END_VAR
TEST('Check_UINT_TO_LWORD_Max');

// @TEST-RUN
converted := TryConvert_UINT_TO_Destination(value, actual);
equal := actual = UINT_TO_LWORD(value);

// @TEST-ASSERT
AssertTrue(Condition := equal, Message := 'Did not convert UINT to LWORD correctly');
AssertTrue(Condition := converted, Message := 'Did not report UINT to LWORD conversion was successful');

TEST_FINISHED();
END_METHOD

METHOD PUBLIC Check_UINT_TO_LWORD_Min
VAR
	value : UINT := DatatypeLimits.UINT_MIN_VALUE;
	actual : LWORD;
	converted : BOOL;
	equal : BOOL;
END_VAR
TEST('Check_UINT_TO_LWORD_Min');

// @TEST-RUN
converted := TryConvert_UINT_TO_Destination(value, actual);
equal := actual = UINT_TO_LWORD(value);

// @TEST-ASSERT
AssertTrue(Condition := equal, Message := 'Did not convert UINT to LWORD correctly');
AssertTrue(Condition := converted, Message := 'Did not report UINT to LWORD conversion was successful');

TEST_FINISHED();
END_METHOD

METHOD PUBLIC Check_UINT_TO_REAL_Max
VAR
	value : UINT := DatatypeLimits.UINT_MAX_VALUE;
	actual : REAL;
	converted : BOOL;
	equal : BOOL;
END_VAR
TEST('Check_UINT_TO_REAL_Max');

// @TEST-RUN
converted := TryConvert_UINT_TO_Destination(value, actual);
equal := actual = UINT_TO_REAL(value);

// @TEST-ASSERT
AssertTrue(Condition := equal, Message := 'Did not convert UINT to REAL correctly');
AssertTrue(Condition := converted, Message := 'Did not report UINT to REAL conversion was successful');

TEST_FINISHED();
END_METHOD

METHOD PUBLIC Check_UINT_TO_REAL_Min
VAR
	value : UINT := DatatypeLimits.UINT_MIN_VALUE;
	actual : REAL;
	converted : BOOL;
	equal : BOOL;
END_VAR
TEST('Check_UINT_TO_REAL_Min');

// @TEST-RUN
converted := TryConvert_UINT_TO_Destination(value, actual);
equal := actual = UINT_TO_REAL(value);

// @TEST-ASSERT
AssertTrue(Condition := equal, Message := 'Did not convert UINT to REAL correctly');
AssertTrue(Condition := converted, Message := 'Did not report UINT to REAL conversion was successful');

TEST_FINISHED();
END_METHOD

METHOD PUBLIC Check_UINT_TO_SINT_Max
VAR
	value : UINT := DatatypeLimits.MAX_VALUE_OF_UINT_WHICH_CAN_BE_HELD_IN_A_SINT;
	actual : SINT;
	converted : BOOL;
	equal : BOOL;
END_VAR
TEST('Check_UINT_TO_SINT_Max');

// @TEST-RUN
converted := TryConvert_UINT_TO_Destination(value, actual);
equal := actual = UINT_TO_SINT(value);

// @TEST-ASSERT
AssertTrue(Condition := equal, Message := 'Did not convert UINT to SINT correctly');
AssertTrue(Condition := converted, Message := 'Did not report UINT to SINT conversion was successful');

TEST_FINISHED();
END_METHOD

METHOD PUBLIC Check_UINT_TO_SINT_Min
VAR
	value : UINT := DatatypeLimits.UINT_MIN_VALUE;
	actual : SINT;
	converted : BOOL;
	equal : BOOL;
END_VAR
TEST('Check_UINT_TO_SINT_Min');

// @TEST-RUN
converted := TryConvert_UINT_TO_Destination(value, actual);
equal := actual = UINT_TO_SINT(value);

// @TEST-ASSERT
AssertTrue(Condition := equal, Message := 'Did not convert UINT to SINT correctly');
AssertTrue(Condition := converted, Message := 'Did not report UINT to SINT conversion was successful');

TEST_FINISHED();
END_METHOD

METHOD PUBLIC Check_UINT_TO_SINT_TooHigh
VAR
	value : UINT := DatatypeLimits.UINT_MAX_VALUE;
	actual : SINT;
	converted : BOOL;
END_VAR
TEST('Check_UINT_TO_SINT_TooHigh');

// @TEST-RUN
converted := TryConvert_UINT_TO_Destination(value, actual);

// @TEST-ASSERT
AssertFalse(Condition := converted, Message := 'Did not report UINT to SINT conversion was prevented');

TEST_FINISHED();
END_METHOD

METHOD PUBLIC Check_UINT_TO_STRING_Max
VAR
	value : UINT := DatatypeLimits.UINT_MAX_VALUE;
	actual : STRING;
	converted : BOOL;
	equal : BOOL;
END_VAR
TEST('Check_UINT_TO_STRING_Max');

// @TEST-RUN
converted := TryConvert_UINT_TO_Destination(value, actual);
equal := actual = UINT_TO_STRING(value);

// @TEST-ASSERT
AssertTrue(Condition := equal, Message := 'Did not convert UINT to STRING correctly');
AssertTrue(Condition := converted, Message := 'Did not report UINT to STRING conversion was successful');

TEST_FINISHED();
END_METHOD

METHOD PUBLIC Check_UINT_TO_STRING_Min
VAR
	value : UINT := DatatypeLimits.UINT_MIN_VALUE;
	actual : STRING;
	converted : BOOL;
	equal : BOOL;
END_VAR
TEST('Check_UINT_TO_STRING_Min');

// @TEST-RUN
converted := TryConvert_UINT_TO_Destination(value, actual);
equal := actual = UINT_TO_STRING(value);

// @TEST-ASSERT
AssertTrue(Condition := equal, Message := 'Did not convert UINT to STRING correctly');
AssertTrue(Condition := converted, Message := 'Did not report UINT to STRING conversion was successful');

TEST_FINISHED();
END_METHOD

METHOD PUBLIC Check_UINT_TO_TIME_Max
VAR
	value : UINT := DatatypeLimits.UINT_MAX_VALUE;
	actual : TIME;
	converted : BOOL;
	equal : BOOL;
END_VAR
TEST('Check_UINT_TO_TIME_Max');

// @TEST-RUN
converted := TryConvert_UINT_TO_Destination(value, actual);
equal := actual = UINT_TO_TIME(value);

// @TEST-ASSERT
AssertTrue(Condition := equal, Message := 'Did not convert UINT to TIME correctly');
AssertTrue(Condition := converted, Message := 'Did not report UINT to TIME conversion was successful');

TEST_FINISHED();
END_METHOD

METHOD PUBLIC Check_UINT_TO_TIME_Min
VAR
	value : UINT := DatatypeLimits.UINT_MIN_VALUE;
	actual : TIME;
	converted : BOOL;
	equal : BOOL;
END_VAR
TEST('Check_UINT_TO_TIME_Min');

// @TEST-RUN
converted := TryConvert_UINT_TO_Destination(value, actual);
equal := actual = UINT_TO_TIME(value);

// @TEST-ASSERT
AssertTrue(Condition := equal, Message := 'Did not convert UINT to TIME correctly');
AssertTrue(Condition := converted, Message := 'Did not report UINT to TIME conversion was successful');

TEST_FINISHED();
END_METHOD

METHOD PUBLIC Check_UINT_TO_TOD_Max
VAR
	value : UINT := DatatypeLimits.UINT_MAX_VALUE;
	actual : TOD;
	converted : BOOL;
	equal : BOOL;
END_VAR
TEST('Check_UINT_TO_TOD_Max');

// @TEST-RUN
converted := TryConvert_UINT_TO_Destination(value, actual);
equal := actual = UINT_TO_TOD(value);

// @TEST-ASSERT
AssertTrue(Condition := equal, Message := 'Did not convert UINT to TOD correctly');
AssertTrue(Condition := converted, Message := 'Did not report UINT to TOD conversion was successful');

TEST_FINISHED();
END_METHOD

METHOD PUBLIC Check_UINT_TO_TOD_Min
VAR
	value : UINT := DatatypeLimits.UINT_MIN_VALUE;
	actual : TOD;
	converted : BOOL;
	equal : BOOL;
END_VAR
TEST('Check_UINT_TO_TOD_Min');

// @TEST-RUN
converted := TryConvert_UINT_TO_Destination(value, actual);
equal := actual = UINT_TO_TOD(value);

// @TEST-ASSERT
AssertTrue(Condition := equal, Message := 'Did not convert UINT to TOD correctly');
AssertTrue(Condition := converted, Message := 'Did not report UINT to TOD conversion was successful');

TEST_FINISHED();
END_METHOD

METHOD PUBLIC Check_UINT_TO_UDINT_Max
VAR
	value : UINT := DatatypeLimits.UINT_MAX_VALUE;
	actual : UDINT;
	converted : BOOL;
	equal : BOOL;
END_VAR
TEST('Check_UINT_TO_UDINT_Max');

// @TEST-RUN
converted := TryConvert_UINT_TO_Destination(value, actual);
equal := actual = UINT_TO_UDINT(value);

// @TEST-ASSERT
AssertTrue(Condition := equal, Message := 'Did not convert UINT to UDINT correctly');
AssertTrue(Condition := converted, Message := 'Did not report UINT to UDINT conversion was successful');

TEST_FINISHED();
END_METHOD

METHOD PUBLIC Check_UINT_TO_UDINT_Min
VAR
	value : UINT := DatatypeLimits.UINT_MIN_VALUE;
	actual : UDINT;
	converted : BOOL;
	equal : BOOL;
END_VAR
TEST('Check_UINT_TO_UDINT_Min');

// @TEST-RUN
converted := TryConvert_UINT_TO_Destination(value, actual);
equal := actual = UINT_TO_UDINT(value);

// @TEST-ASSERT
AssertTrue(Condition := equal, Message := 'Did not convert UINT to UDINT correctly');
AssertTrue(Condition := converted, Message := 'Did not report UINT to UDINT conversion was successful');

TEST_FINISHED();
END_METHOD

METHOD PUBLIC Check_UINT_TO_UINT_Max
VAR
	value : UINT := DatatypeLimits.UINT_MAX_VALUE;
	actual : UINT;
	converted : BOOL;
	equal : BOOL;
END_VAR
TEST('Check_UINT_TO_UINT_Max');

// @TEST-RUN
converted := TryConvert_UINT_TO_Destination(value, actual);
equal := actual = value;

// @TEST-ASSERT
AssertTrue(Condition := equal, Message := 'Did not convert UINT to UINT correctly');
AssertTrue(Condition := converted, Message := 'Did not report UINT to UINT conversion was successful');

TEST_FINISHED();
END_METHOD

METHOD PUBLIC Check_UINT_TO_UINT_Min
VAR
	value : UINT := DatatypeLimits.UINT_MIN_VALUE;
	actual : UINT;
	converted : BOOL;
	equal : BOOL;
END_VAR
TEST('Check_UINT_TO_UINT_Min');

// @TEST-RUN
converted := TryConvert_UINT_TO_Destination(value, actual);
equal := actual = value;

// @TEST-ASSERT
AssertTrue(Condition := equal, Message := 'Did not convert UINT to UINT correctly');
AssertTrue(Condition := converted, Message := 'Did not report UINT to UINT conversion was successful');

TEST_FINISHED();
END_METHOD

METHOD PUBLIC Check_UINT_TO_ULINT_Max
VAR
	value : UINT := DatatypeLimits.UINT_MAX_VALUE;
	actual : ULINT;
	converted : BOOL;
	equal : BOOL;
END_VAR
TEST('Check_UINT_TO_ULINT_Max');

// @TEST-RUN
converted := TryConvert_UINT_TO_Destination(value, actual);
equal := actual = UINT_TO_ULINT(value);

// @TEST-ASSERT
AssertTrue(Condition := equal, Message := 'Did not convert UINT to ULINT correctly');
AssertTrue(Condition := converted, Message := 'Did not report UINT to ULINT conversion was successful');

TEST_FINISHED();
END_METHOD

METHOD PUBLIC Check_UINT_TO_ULINT_Min
VAR
	value : UINT := DatatypeLimits.UINT_MIN_VALUE;
	actual : ULINT;
	converted : BOOL;
	equal : BOOL;
END_VAR
TEST('Check_UINT_TO_ULINT_Min');

// @TEST-RUN
converted := TryConvert_UINT_TO_Destination(value, actual);
equal := actual = UINT_TO_ULINT(value);

// @TEST-ASSERT
AssertTrue(Condition := equal, Message := 'Did not convert UINT to ULINT correctly');
AssertTrue(Condition := converted, Message := 'Did not report UINT to ULINT conversion was successful');

TEST_FINISHED();
END_METHOD

METHOD PUBLIC Check_UINT_TO_USINT_Max
VAR
	value : UINT := DatatypeLimits.MAX_VALUE_OF_UINT_WHICH_CAN_BE_HELD_IN_A_USINT;
	actual : USINT;
	converted : BOOL;
	equal : BOOL;
END_VAR
TEST('Check_UINT_TO_USINT_Max');

// @TEST-RUN
converted := TryConvert_UINT_TO_Destination(value, actual);
equal := actual = UINT_TO_USINT(value);

// @TEST-ASSERT
AssertTrue(Condition := equal, Message := 'Did not convert UINT to USINT correctly');
AssertTrue(Condition := converted, Message := 'Did not report UINT to USINT conversion was successful');

TEST_FINISHED();
END_METHOD

METHOD PUBLIC Check_UINT_TO_USINT_Min
VAR
	value : UINT := DatatypeLimits.UINT_MIN_VALUE;
	actual : USINT;
	converted : BOOL;
	equal : BOOL;
END_VAR
TEST('Check_UINT_TO_USINT_Min');

// @TEST-RUN
converted := TryConvert_UINT_TO_Destination(value, actual);
equal := actual = UINT_TO_USINT(value);

// @TEST-ASSERT
AssertTrue(Condition := equal, Message := 'Did not convert UINT to USINT correctly');
AssertTrue(Condition := converted, Message := 'Did not report UINT to USINT conversion was successful');

TEST_FINISHED();
END_METHOD

METHOD PUBLIC Check_UINT_TO_USINT_TooHigh
VAR
	value : UINT := DatatypeLimits.UINT_MAX_VALUE;
	actual : USINT;
	converted : BOOL;
END_VAR
TEST('Check_UINT_TO_USINT_TooHigh');

// @TEST-RUN
converted := TryConvert_UINT_TO_Destination(value, actual);

// @TEST-ASSERT
AssertFalse(Condition := converted, Message := 'Did not report UINT to USINT conversion was prevented');

TEST_FINISHED();
END_METHOD

METHOD PUBLIC Check_UINT_TO_WORD_Max
VAR
	value : UINT := DatatypeLimits.UINT_MAX_VALUE;
	actual : WORD;
	converted : BOOL;
	equal : BOOL;
END_VAR
TEST('Check_UINT_TO_WORD_Max');

// @TEST-RUN
converted := TryConvert_UINT_TO_Destination(value, actual);
equal := actual = UINT_TO_WORD(value);

// @TEST-ASSERT
AssertTrue(Condition := equal, Message := 'Did not convert UINT to WORD correctly');
AssertTrue(Condition := converted, Message := 'Did not report UINT to WORD conversion was successful');

TEST_FINISHED();
END_METHOD

METHOD PUBLIC Check_UINT_TO_WORD_Min
VAR
	value : UINT := DatatypeLimits.UINT_MIN_VALUE;
	actual : WORD;
	converted : BOOL;
	equal : BOOL;
END_VAR
TEST('Check_UINT_TO_WORD_Min');

// @TEST-RUN
converted := TryConvert_UINT_TO_Destination(value, actual);
equal := actual = UINT_TO_WORD(value);

// @TEST-ASSERT
AssertTrue(Condition := equal, Message := 'Did not convert UINT to WORD correctly');
AssertTrue(Condition := converted, Message := 'Did not report UINT to WORD conversion was successful');

TEST_FINISHED();
END_METHOD

END_FUNCTION_BLOCK

// ---- mobject-converters/Tests/WORD_TO_TestSuite.TcPOU
FUNCTION_BLOCK PUBLIC WORD_TO_TestSuite EXTENDS TcUnit.FB_TestSuite
VAR
END_VAR

